LIN {X 0,Y 573.279,Z 329.697,A -85,B 0,C 180,E1 -2325.807,E2 -2325.807} C_VEL
LIN {X 0,Y 573.268,Z 329.699,A -85,B 0,C 180,E1 -2328.745,E2 -2328.745} C_VEL
LIN {X 0,Y 573.26,Z 329.706,A -85,B 0,C 180,E1 -2331.54,E2 -2331.54} C_VEL
LIN {X 0,Y 573.246,Z 329.702,A -85,B 0,C 180,E1 -2333.665,E2 -2333.665} C_VEL
LIN {X 0,Y 573.226,Z 329.704,A -85,B 0,C 180,E1 -2335.781,E2 -2335.781} C_VEL
LIN {X 0,Y 573.314,Z 329.695,A -85,B 0,C 180,E1 -2337.893,E2 -2337.893} C_VEL
LIN {X 0,Y 573.335,Z 329.689,A -85,B 0,C 180,E1 -2340.702,E2 -2340.702} C_VEL
LIN {X 0,Y 573.237,Z 329.705,A -85,B 0,C 180,E1 -2343.515,E2 -2343.515} C_VEL
LIN {X 0,Y 573.295,Z 329.695,A -85,B 0,C 180,E1 -2345.628,E2 -2345.628} C_VEL
LIN {X 0,Y 573.277,Z 329.698,A -85,B 0,C 180,E1 -2347.75,E2 -2347.75} C_VEL
LIN {X 0,Y 573.271,Z 329.698,A -85,B 0,C 180,E1 -2350.597,E2 -2350.597} C_VEL
LIN {X 0,Y 573.269,Z 329.699,A -85,B 0,C 180,E1 -2352.749,E2 -2352.749} C_VEL
LIN {X 0,Y 573.241,Z 329.707,A -85,B 0,C 180,E1 -2354.92,E2 -2354.92} C_VEL
LIN {X 0,Y 573.249,Z 329.701,A -85,B 0,C 180,E1 -2357.848,E2 -2357.848} C_VEL
LIN {X 0,Y 573.246,Z 329.708,A -85,B 0,C 180,E1 -2360.077,E2 -2360.077} C_VEL
LIN {X 0,Y 573.24,Z 329.703,A -85,B 0,C 180,E1 -2362.338,E2 -2362.338} C_VEL
LIN {X 0,Y 573.255,Z 329.699,A -85,B 0,C 180,E1 -2364.389,E2 -2364.389} C_VEL
LIN {X 0,Y 572.629,Z 329.784,A -85,B 0,C 180,E1 -2364.976,E2 -2364.976} C_VEL
LIN {X 0,Y 569.786,Z 330.135,A -85,B 0,C 180,E1 -2365.927,E2 -2365.927} C_VEL
LIN {X 0,Y 567.354,Z 330.441,A -85,B 0,C 180,E1 -2366.693,E2 -2366.693} C_VEL
LIN {X 0,Y 566.298,Z 330.568,A -85,B 0,C 180,E1 -2367.284,E2 -2367.284} C_VEL
LIN {X 0,Y 566.208,Z 330.578,A -85,B 0,C 180,E1 -2367.484,E2 -2367.484} C_VEL
LIN {X 0,Y 566.206,Z 330.58,A -85,B 0,C 180,E1 -2369.769,E2 -2369.769} C_VEL
LIN {X 0,Y 566.207,Z 330.579,A -85,B 0,C 180,E1 -2372.43,E2 -2372.43} C_VEL
LIN {X 0,Y 566.186,Z 330.585,A -85,B 0,C 180,E1 -2374.99,E2 -2374.99} C_VEL
LIN {X 0,Y 566.2,Z 330.58,A -85,B 0,C 180,E1 -2377.461,E2 -2377.461} C_VEL
LIN {X 0,Y 566.211,Z 330.584,A -85,B 0,C 180,E1 -2380.199,E2 -2380.199} C_VEL
LIN {X 0,Y 566.205,Z 330.579,A -85,B 0,C 180,E1 -2383.054,E2 -2383.054} C_VEL
LIN {X 0,Y 566.203,Z 330.58,A -85,B 0,C 180,E1 -2386.049,E2 -2386.049} C_VEL
LIN {X 0,Y 566.186,Z 330.586,A -85,B 0,C 180,E1 -2388.861,E2 -2388.861} C_VEL
LIN {X 0,Y 566.274,Z 330.749,A -85,B 0,C 180,E1 -2391.305,E2 -2391.305} C_VEL
LIN {X 0,Y 566.32,Z 335.336,A -85,B 0,C 180,E1 -2393.77,E2 -2393.77} C_VEL
LIN {X 0,Y 566.259,Z 339.965,A -85,B 0,C 180,E1 -2396.259,E2 -2396.259} C_VEL
LIN {X 0,Y 566.185,Z 344.997,A -85,B 0,C 180,E1 -2398.925,E2 -2398.925} C_VEL
LIN {X 0,Y 566.125,Z 350.67,A -85,B 0,C 180,E1 -2401.852,E2 -2401.852} C_VEL
LIN {X 0,Y 566.061,Z 355.376,A -85,B 0,C 180,E1 -2404.243,E2 -2404.243} C_VEL
LIN {X 0,Y 566.048,Z 360.406,A -85,B 0,C 180,E1 -2406.748,E2 -2406.748} C_VEL
LIN {X 0,Y 566.016,Z 364.889,A -85,B 0,C 180,E1 -2408.895,E2 -2408.895} C_VEL
LIN {X 0,Y 565.984,Z 371.303,A -85,B 0,C 180,E1 -2411.915,E2 -2411.915} C_VEL
LIN {X 0,Y 565.961,Z 377.468,A -85,B 0,C 180,E1 -2414.769,E2 -2414.769} C_VEL
LIN {X 0,Y 567.384,Z 385.385,A -85,B 0,C 180,E1 -2414.949,E2 -2414.949} C_VEL
LIN {X 0,Y 567.258,Z 399.805,A -85,B 0,C 180,E1 -2415.313,E2 -2415.313} C_VEL
LIN {X 0,Y 567.093,Z 414.1,A -85,B 0,C 180,E1 -2415.832,E2 -2415.832} C_VEL
LIN {X 0,Y 566.914,Z 427.265,A -85,B 0,C 180,E1 -2416.468,E2 -2416.468} C_VEL
LIN {X 0,Y 566.715,Z 439.211,A -85,B 0,C 180,E1 -2417.193,E2 -2417.193} C_VEL
LIN {X 0,Y 566.536,Z 451.291,A -85,B 0,C 180,E1 -2418.098,E2 -2418.098} C_VEL
LIN {X 0,Y 566.399,Z 462.502,A -85,B 0,C 180,E1 -2419.126,E2 -2419.126} C_VEL
LIN {X 0,Y 566.202,Z 471.968,A -85,B 0,C 180,E1 -2420.173,E2 -2420.173} C_VEL
LIN {X 0,Y 566.123,Z 480.099,A -85,B 0,C 180,E1 -2421.253,E2 -2421.253} C_VEL
LIN {X 0,Y 566.016,Z 487.881,A -85,B 0,C 180,E1 -2422.509,E2 -2422.509} C_VEL
LIN {X 0,Y 565.945,Z 493.323,A -85,B 0,C 180,E1 -2423.583,E2 -2423.583} C_VEL
LIN {X 0,Y 565.928,Z 497.801,A -85,B 0,C 180,E1 -2424.656,E2 -2424.656} C_VEL
LIN {X 0,Y 565.957,Z 501.311,A -85,B 0,C 180,E1 -2425.727,E2 -2425.727} C_VEL
LIN {X 0,Y 565.875,Z 504.742,A -85,B 0,C 180,E1 -2427.152,E2 -2427.152} C_VEL
LIN {X 0,Y 565.844,Z 506.784,A -85,B 0,C 180,E1 -2428.577,E2 -2428.577} C_VEL
LIN {X 0,Y 565.838,Z 507.496,A -85,B 0,C 180,E1 -2430,E2 -2430} C_VEL
LIN {X 0,Y 565.841,Z 506.881,A -85,B 0,C 180,E1 -2431.424,E2 -2431.424} C_VEL
LIN {X 0,Y 565.873,Z 504.925,A -85,B 0,C 180,E1 -2432.848,E2 -2432.848} C_VEL
LIN {X 0,Y 565.958,Z 501.577,A -85,B 0,C 180,E1 -2434.273,E2 -2434.273} C_VEL
LIN {X 0,Y 565.983,Z 496.745,A -85,B 0,C 180,E1 -2435.701,E2 -2435.701} C_VEL
LIN {X 0,Y 565.981,Z 490.281,A -85,B 0,C 180,E1 -2437.133,E2 -2437.133} C_VEL
LIN {X 0,Y 566.093,Z 483.08,A -85,B 0,C 180,E1 -2438.388,E2 -2438.388} C_VEL
LIN {X 0,Y 566.172,Z 475.539,A -85,B 0,C 180,E1 -2439.467,E2 -2439.467} C_VEL
LIN {X 0,Y 566.29,Z 466.484,A -85,B 0,C 180,E1 -2440.548,E2 -2440.548} C_VEL
LIN {X 0,Y 566.487,Z 457.47,A -85,B 0,C 180,E1 -2441.449,E2 -2441.449} C_VEL
LIN {X 0,Y 566.626,Z 446.716,A -85,B 0,C 180,E1 -2442.354,E2 -2442.354} C_VEL
LIN {X 0,Y 566.767,Z 434.955,A -85,B 0,C 180,E1 -2443.171,E2 -2443.171} C_VEL
LIN {X 0,Y 567.011,Z 421.978,A -85,B 0,C 180,E1 -2443.896,E2 -2443.896} C_VEL
LIN {X 0,Y 567.185,Z 409.289,A -85,B 0,C 180,E1 -2444.451,E2 -2444.451} C_VEL
LIN {X 0,Y 567.306,Z 395.024,A -85,B 0,C 180,E1 -2444.918,E2 -2444.918} C_VEL
LIN {X 0,Y 567.183,Z 383.552,A -85,B 0,C 180,E1 -2445.183,E2 -2445.183} C_VEL
LIN {X 0,Y 565.932,Z 377.463,A -85,B 0,C 180,E1 -2445.324,E2 -2445.324} C_VEL
LIN {X 0,Y 565.976,Z 371.496,A -85,B 0,C 180,E1 -2448.086,E2 -2448.086} C_VEL
LIN {X 0,Y 566.018,Z 365.078,A -85,B 0,C 180,E1 -2451.105,E2 -2451.105} C_VEL
LIN {X 0,Y 566.039,Z 358.692,A -85,B 0,C 180,E1 -2454.188,E2 -2454.188} C_VEL
LIN {X 0,Y 566.084,Z 353.819,A -85,B 0,C 180,E1 -2456.634,E2 -2456.634} C_VEL
LIN {X 0,Y 566.132,Z 349.269,A -85,B 0,C 180,E1 -2458.957,E2 -2458.957} C_VEL
LIN {X 0,Y 566.192,Z 344.506,A -85,B 0,C 180,E1 -2461.422,E2 -2461.422} C_VEL
LIN {X 0,Y 566.258,Z 339.744,A -85,B 0,C 180,E1 -2463.953,E2 -2463.953} C_VEL
LIN {X 0,Y 566.314,Z 334.886,A -85,B 0,C 180,E1 -2466.562,E2 -2466.562} C_VEL
LIN {X 0,Y 566.225,Z 330.582,A -85,B 0,C 180,E1 -2468.893,E2 -2468.893} C_VEL
LIN {X 0,Y 566.193,Z 330.583,A -85,B 0,C 180,E1 -2471.861,E2 -2471.861} C_VEL
LIN {X 0,Y 566.203,Z 330.579,A -85,B 0,C 180,E1 -2474.036,E2 -2474.036} C_VEL
LIN {X 0,Y 566.206,Z 330.578,A -85,B 0,C 180,E1 -2477.083,E2 -2477.083} C_VEL
LIN {X 0,Y 566.221,Z 330.577,A -85,B 0,C 180,E1 -2480.314,E2 -2480.314} C_VEL
LIN {X 0,Y 566.205,Z 330.582,A -85,B 0,C 180,E1 -2483.43,E2 -2483.43} C_VEL
LIN {X 0,Y 566.218,Z 330.58,A -85,B 0,C 180,E1 -2486.266,E2 -2486.266} C_VEL
LIN {X 0,Y 566.196,Z 330.58,A -85,B 0,C 180,E1 -2488.924,E2 -2488.924} C_VEL
LIN {X 0,Y 566.218,Z 330.58,A -85,B 0,C 180,E1 -2491.858,E2 -2491.858} C_VEL
LIN {X 0,Y 566.215,Z 330.577,A -85,B 0,C 180,E1 -2494.251,E2 -2494.251} C_VEL
LIN {X 0,Y 566.179,Z 330.588,A -85,B 0,C 180,E1 -2496.718,E2 -2496.718} C_VEL
LIN {X 0,Y 566.213,Z 330.579,A -85,B 0,C 180,E1 -2499.663,E2 -2499.663} C_VEL
LIN {X 0,Y 566.206,Z 330.578,A -85,B 0,C 180,E1 -2502.668,E2 -2502.668} C_VEL
LIN {X 0,Y 566.236,Z 330.575,A -85,B 0,C 180,E1 -2505.627,E2 -2505.627} C_VEL
LIN {X 0,Y 566.242,Z 330.577,A -85,B 0,C 180,E1 -2508.675,E2 -2508.675} C_VEL
LIN {X 0,Y 566.212,Z 330.58,A -85,B 0,C 180,E1 -2511.434,E2 -2511.434} C_VEL
LIN {X 0,Y 566.263,Z 330.571,A -85,B 0,C 180,E1 -2514.302,E2 -2514.302} C_VEL
LIN {X 0,Y 566.28,Z 330.569,A -85,B 0,C 180,E1 -2517.866,E2 -2517.866} C_VEL
LIN {X 0,Y 566.307,Z 330.566,A -85,B 0,C 180,E1 -2520.711,E2 -2520.711} C_VEL
LIN {X 0,Y 566.277,Z 330.57,A -85,B 0,C 180,E1 -2522.845,E2 -2522.845} C_VEL
LIN {X 0,Y 566.263,Z 330.572,A -85,B 0,C 180,E1 -2525.698,E2 -2525.698} C_VEL
LIN {X 0,Y 566.212,Z 330.584,A -85,B 0,C 180,E1 -2528.566,E2 -2528.566} C_VEL
LIN {X 0,Y 566.249,Z 330.574,A -85,B 0,C 180,E1 -2531.454,E2 -2531.454} C_VEL
LIN {X 0,Y 566.241,Z 330.574,A -85,B 0,C 180,E1 -2534.506,E2 -2534.506} C_VEL
LIN {X 0,Y 566.206,Z 330.581,A -85,B 0,C 180,E1 -2537.331,E2 -2537.331} C_VEL
LIN {X 0,Y 566.213,Z 330.585,A -85,B 0,C 180,E1 -2540.337,E2 -2540.337} C_VEL
LIN {X 0,Y 566.195,Z 330.583,A -85,B 0,C 180,E1 -2543.403,E2 -2543.403} C_VEL
LIN {X 0,Y 566.219,Z 330.579,A -85,B 0,C 180,E1 -2545.749,E2 -2545.749} C_VEL
LIN {X 0,Y 566.208,Z 330.579,A -85,B 0,C 180,E1 -2548.202,E2 -2548.202} C_VEL
LIN {X 0,Y 566.195,Z 330.58,A -85,B 0,C 180,E1 -2551.076,E2 -2551.076} C_VEL
LIN {X 0,Y 566.217,Z 330.584,A -85,B 0,C 180,E1 -2553.734,E2 -2553.734} C_VEL
LIN {X 0,Y 566.22,Z 330.578,A -85,B 0,C 180,E1 -2556.568,E2 -2556.568} C_VEL
LIN {X 0,Y 566.22,Z 330.576,A -85,B 0,C 180,E1 -2559.686,E2 -2559.686} C_VEL
LIN {X 0,Y 566.214,Z 330.584,A -85,B 0,C 180,E1 -2562.087,E2 -2562.087} C_VEL
LIN {X 0,Y 566.173,Z 330.584,A -85,B 0,C 180,E1 -2565.036,E2 -2565.036} C_VEL
LIN {X 0,Y 566.218,Z 330.578,A -85,B 0,C 180,E1 -2567.913,E2 -2567.913} C_VEL
LIN {X 0,Y 566.217,Z 330.583,A -85,B 0,C 180,E1 -2570.726,E2 -2570.726} C_VEL
LIN {X 0,Y 566.247,Z 330.784,A -85,B 0,C 180,E1 -2573.534,E2 -2573.534} C_VEL
LIN {X 0,Y 567.061,Z 335.097,A -85,B 0,C 180,E1 -2574.883,E2 -2574.883} C_VEL
LIN {X 0,Y 566.991,Z 342.231,A -85,B 0,C 180,E1 -2576.948,E2 -2576.948} C_VEL
LIN {X 0,Y 566.836,Z 352.746,A -85,B 0,C 180,E1 -2579.858,E2 -2579.858} C_VEL
LIN {X 0,Y 566.665,Z 363.294,A -85,B 0,C 180,E1 -2582.684,E2 -2582.684} C_VEL
LIN {X 0,Y 566.483,Z 373.873,A -85,B 0,C 180,E1 -2585.442,E2 -2585.442} C_VEL
LIN {X 0,Y 566.404,Z 382.902,A -85,B 0,C 180,E1 -2587.762,E2 -2587.762} C_VEL
LIN {X 0,Y 566.295,Z 394.128,A -85,B 0,C 180,E1 -2590.595,E2 -2590.595} C_VEL
LIN {X 0,Y 566.236,Z 400.283,A -85,B 0,C 180,E1 -2592.128,E2 -2592.128} C_VEL
LIN {X 0,Y 567.998,Z 408.781,A -85,B 0,C 180,E1 -2592.315,E2 -2592.315} C_VEL
LIN {X 0,Y 567.88,Z 424.081,A -85,B 0,C 180,E1 -2592.628,E2 -2592.628} C_VEL
LIN {X 0,Y 567.684,Z 439.2,A -85,B 0,C 180,E1 -2593.086,E2 -2593.086} C_VEL
LIN {X 0,Y 567.454,Z 452.815,A -85,B 0,C 180,E1 -2593.634,E2 -2593.634} C_VEL
LIN {X 0,Y 567.232,Z 467.096,A -85,B 0,C 180,E1 -2594.366,E2 -2594.366} C_VEL
LIN {X 0,Y 566.953,Z 480.511,A -85,B 0,C 180,E1 -2595.216,E2 -2595.216} C_VEL
LIN {X 0,Y 566.738,Z 493.158,A -85,B 0,C 180,E1 -2596.189,E2 -2596.189} C_VEL
LIN {X 0,Y 566.546,Z 504.968,A -85,B 0,C 180,E1 -2597.28,E2 -2597.28} C_VEL
LIN {X 0,Y 566.343,Z 514.901,A -85,B 0,C 180,E1 -2598.366,E2 -2598.366} C_VEL
LIN {X 0,Y 566.204,Z 524.619,A -85,B 0,C 180,E1 -2599.631,E2 -2599.631} C_VEL
LIN {X 0,Y 566.079,Z 532.721,A -85,B 0,C 180,E1 -2600.892,E2 -2600.892} C_VEL
LIN {X 0,Y 566.014,Z 539.424,A -85,B 0,C 180,E1 -2602.15,E2 -2602.15} C_VEL
LIN {X 0,Y 565.943,Z 545.606,A -85,B 0,C 180,E1 -2603.583,E2 -2603.583} C_VEL
LIN {X 0,Y 565.867,Z 550.385,A -85,B 0,C 180,E1 -2605.012,E2 -2605.012} C_VEL
LIN {X 0,Y 565.909,Z 553.889,A -85,B 0,C 180,E1 -2606.44,E2 -2606.44} C_VEL
LIN {X 0,Y 565.839,Z 556.192,A -85,B 0,C 180,E1 -2607.864,E2 -2607.864} C_VEL
LIN {X 0,Y 565.839,Z 557.349,A -85,B 0,C 180,E1 -2609.288,E2 -2609.288} C_VEL
LIN {X 0,Y 565.839,Z 557.349,A -85,B 0,C 180,E1 -2610.712,E2 -2610.712} C_VEL
LIN {X 0,Y 565.839,Z 556.191,A -85,B 0,C 180,E1 -2612.135,E2 -2612.135} C_VEL
LIN {X 0,Y 565.909,Z 553.887,A -85,B 0,C 180,E1 -2613.56,E2 -2613.56} C_VEL
LIN {X 0,Y 565.866,Z 550.385,A -85,B 0,C 180,E1 -2614.988,E2 -2614.988} C_VEL
LIN {X 0,Y 565.942,Z 545.609,A -85,B 0,C 180,E1 -2616.417,E2 -2616.417} C_VEL
LIN {X 0,Y 566.014,Z 539.423,A -85,B 0,C 180,E1 -2617.85,E2 -2617.85} C_VEL
LIN {X 0,Y 566.071,Z 531.648,A -85,B 0,C 180,E1 -2619.288,E2 -2619.288} C_VEL
LIN {X 0,Y 566.24,Z 523.369,A -85,B 0,C 180,E1 -2620.549,E2 -2620.549} C_VEL
LIN {X 0,Y 566.367,Z 513.391,A -85,B 0,C 180,E1 -2621.815,E2 -2621.815} C_VEL
LIN {X 0,Y 566.586,Z 503.188,A -85,B 0,C 180,E1 -2622.901,E2 -2622.901} C_VEL
LIN {X 0,Y 566.763,Z 491.018,A -85,B 0,C 180,E1 -2623.993,E2 -2623.993} C_VEL
LIN {X 0,Y 567.041,Z 478.339,A -85,B 0,C 180,E1 -2624.936,E2 -2624.936} C_VEL
LIN {X 0,Y 567.266,Z 465.514,A -85,B 0,C 180,E1 -2625.725,E2 -2625.725} C_VEL
LIN {X 0,Y 567.494,Z 450.83,A -85,B 0,C 180,E1 -2626.457,E2 -2626.457} C_VEL
LIN {X 0,Y 567.721,Z 436.613,A -85,B 0,C 180,E1 -2627.005,E2 -2627.005} C_VEL
LIN {X 0,Y 567.869,Z 422.051,A -85,B 0,C 180,E1 -2627.424,E2 -2627.424} C_VEL
LIN {X 0,Y 567.893,Z 407.611,A -85,B 0,C 180,E1 -2627.706,E2 -2627.706} C_VEL
LIN {X 0,Y 566.243,Z 400.314,A -85,B 0,C 180,E1 -2627.864,E2 -2627.864} C_VEL
LIN {X 0,Y 566.331,Z 388.922,A -85,B 0,C 180,E1 -2630.712,E2 -2630.712} C_VEL
LIN {X 0,Y 566.488,Z 376.883,A -85,B 0,C 180,E1 -2633.779,E2 -2633.779} C_VEL
LIN {X 0,Y 566.614,Z 365.5,A -85,B 0,C 180,E1 -2636.741,E2 -2636.741} C_VEL
LIN {X 0,Y 566.755,Z 355.701,A -85,B 0,C 180,E1 -2639.329,E2 -2639.329} C_VEL
LIN {X 0,Y 566.975,Z 345.213,A -85,B 0,C 180,E1 -2642.209,E2 -2642.209} C_VEL
LIN {X 0,Y 567.084,Z 336.315,A -85,B 0,C 180,E1 -2644.757,E2 -2644.757} C_VEL
LIN {X 0,Y 566.225,Z 330.582,A -85,B 0,C 180,E1 -2646.568,E2 -2646.568} C_VEL
LIN {X 0,Y 566.217,Z 330.583,A -85,B 0,C 180,E1 -2649.686,E2 -2649.686} C_VEL
LIN {X 0,Y 566.217,Z 330.578,A -85,B 0,C 180,E1 -2652.087,E2 -2652.087} C_VEL
LIN {X 0,Y 566.171,Z 330.585,A -85,B 0,C 180,E1 -2655.037,E2 -2655.037} C_VEL
LIN {X 0,Y 566.215,Z 330.579,A -85,B 0,C 180,E1 -2658.137,E2 -2658.137} C_VEL
LIN {X 0,Y 566.225,Z 330.578,A -85,B 0,C 180,E1 -2660.727,E2 -2660.727} C_VEL
LIN {X 0,Y 566.222,Z 330.577,A -85,B 0,C 180,E1 -2663.784,E2 -2663.784} C_VEL
LIN {X 0,Y 566.216,Z 330.584,A -85,B 0,C 180,E1 -2666.266,E2 -2666.266} C_VEL
LIN {X 0,Y 566.194,Z 330.581,A -85,B 0,C 180,E1 -2668.924,E2 -2668.924} C_VEL
LIN {X 0,Y 566.215,Z 330.578,A -85,B 0,C 180,E1 -2671.858,E2 -2671.858} C_VEL
LIN {X 0,Y 566.218,Z 330.579,A -85,B 0,C 180,E1 -2674.251,E2 -2674.251} C_VEL
LIN {X 0,Y 566.196,Z 330.582,A -85,B 0,C 180,E1 -2676.714,E2 -2676.714} C_VEL
LIN {X 0,Y 566.212,Z 330.583,A -85,B 0,C 180,E1 -2679.663,E2 -2679.663} C_VEL
LIN {X 0,Y 566.205,Z 330.58,A -85,B 0,C 180,E1 -2682.669,E2 -2682.669} C_VEL
LIN {X 0,Y 566.24,Z 330.574,A -85,B 0,C 180,E1 -2685.627,E2 -2685.627} C_VEL
LIN {X 0,Y 566.24,Z 330.575,A -85,B 0,C 180,E1 -2688.676,E2 -2688.676} C_VEL
LIN {X 0,Y 566.211,Z 330.584,A -85,B 0,C 180,E1 -2691.434,E2 -2691.434} C_VEL
LIN {X 0,Y 566.263,Z 330.571,A -85,B 0,C 180,E1 -2694.302,E2 -2694.302} C_VEL
LIN {X 0,Y 566.285,Z 330.57,A -85,B 0,C 180,E1 -2697.866,E2 -2697.866} C_VEL
LIN {X 0,Y 566.306,Z 330.565,A -85,B 0,C 180,E1 -2700.711,E2 -2700.711} C_VEL
LIN {X 0,Y 566.277,Z 330.571,A -85,B 0,C 180,E1 -2702.846,E2 -2702.846} C_VEL
LIN {X 0,Y 566.263,Z 330.571,A -85,B 0,C 180,E1 -2705.698,E2 -2705.698} C_VEL
LIN {X 0,Y 566.211,Z 330.581,A -85,B 0,C 180,E1 -2708.566,E2 -2708.566} C_VEL
LIN {X 0,Y 566.248,Z 330.577,A -85,B 0,C 180,E1 -2711.454,E2 -2711.454} C_VEL
LIN {X 0,Y 566.24,Z 330.575,A -85,B 0,C 180,E1 -2714.506,E2 -2714.506} C_VEL
LIN {X 0,Y 566.205,Z 330.578,A -85,B 0,C 180,E1 -2717.332,E2 -2717.332} C_VEL
LIN {X 0,Y 566.212,Z 330.58,A -85,B 0,C 180,E1 -2720.337,E2 -2720.337} C_VEL
LIN {X 0,Y 566.194,Z 330.587,A -85,B 0,C 180,E1 -2723.404,E2 -2723.404} C_VEL
LIN {X 0,Y 566.214,Z 330.578,A -85,B 0,C 180,E1 -2725.749,E2 -2725.749} C_VEL
LIN {X 0,Y 566.208,Z 330.578,A -85,B 0,C 180,E1 -2727.484,E2 -2727.484} C_VEL
LIN {X 0,Y 565.528,Z 330.666,A -85,B 0,C 180,E1 -2728.078,E2 -2728.078} C_VEL
LIN {X 0,Y 562.662,Z 331.023,A -85,B 0,C 180,E1 -2729.041,E2 -2729.041} C_VEL
LIN {X 0,Y 560.252,Z 331.324,A -85,B 0,C 180,E1 -2729.817,E2 -2729.817} C_VEL
LIN {X 0,Y 559.225,Z 331.452,A -85,B 0,C 180,E1 -2730.416,E2 -2730.416} C_VEL
LIN {X 0,Y 559.144,Z 331.459,A -85,B 0,C 180,E1 -2730.618,E2 -2730.618} C_VEL
LIN {X 0,Y 559.17,Z 331.461,A -85,B 0,C 180,E1 -2733.575,E2 -2733.575} C_VEL
LIN {X 0,Y 559.151,Z 331.459,A -85,B 0,C 180,E1 -2736.445,E2 -2736.445} C_VEL
LIN {X 0,Y 559.179,Z 331.456,A -85,B 0,C 180,E1 -2738.934,E2 -2738.934} C_VEL
LIN {X 0,Y 559.167,Z 331.461,A -85,B 0,C 180,E1 -2741.77,E2 -2741.77} C_VEL
LIN {X 0,Y 559.144,Z 331.46,A -85,B 0,C 180,E1 -2744.739,E2 -2744.739} C_VEL
LIN {X 0,Y 559.181,Z 331.455,A -85,B 0,C 180,E1 -2747.863,E2 -2747.863} C_VEL
LIN {X 0,Y 559.222,Z 331.589,A -85,B 0,C 180,E1 -2751.186,E2 -2751.186} C_VEL
LIN {X 0,Y 559.287,Z 336.402,A -85,B 0,C 180,E1 -2753.8,E2 -2753.8} C_VEL
LIN {X 0,Y 559.207,Z 341.235,A -85,B 0,C 180,E1 -2756.428,E2 -2756.428} C_VEL
LIN {X 0,Y 559.149,Z 346.007,A -85,B 0,C 180,E1 -2758.98,E2 -2758.98} C_VEL
LIN {X 0,Y 559.073,Z 352.333,A -85,B 0,C 180,E1 -2762.282,E2 -2762.282} C_VEL
LIN {X 0,Y 559.019,Z 357.368,A -85,B 0,C 180,E1 -2764.849,E2 -2764.849} C_VEL
LIN {X 0,Y 558.948,Z 363.315,A -85,B 0,C 180,E1 -2767.839,E2 -2767.839} C_VEL
LIN {X 0,Y 558.908,Z 369.701,A -85,B 0,C 180,E1 -2770.917,E2 -2770.917} C_VEL
LIN {X 0,Y 558.884,Z 374.512,A -85,B 0,C 180,E1 -2773.188,E2 -2773.188} C_VEL
LIN {X 0,Y 558.882,Z 377.469,A -85,B 0,C 180,E1 -2774.571,E2 -2774.571} C_VEL
LIN {X 0,Y 560.522,Z 386.231,A -85,B 0,C 180,E1 -2774.777,E2 -2774.777} C_VEL
LIN {X 0,Y 560.388,Z 400.196,A -85,B 0,C 180,E1 -2775.14,E2 -2775.14} C_VEL
LIN {X 0,Y 560.21,Z 414.115,A -85,B 0,C 180,E1 -2775.654,E2 -2775.654} C_VEL
LIN {X 0,Y 560,Z 427.276,A -85,B 0,C 180,E1 -2776.297,E2 -2776.297} C_VEL
LIN {X 0,Y 559.76,Z 439.219,A -85,B 0,C 180,E1 -2777.031,E2 -2777.031} C_VEL
LIN {X 0,Y 559.558,Z 451.296,A -85,B 0,C 180,E1 -2777.947,E2 -2777.947} C_VEL
LIN {X 0,Y 559.417,Z 461.299,A -85,B 0,C 180,E1 -2778.864,E2 -2778.864} C_VEL
LIN {X 0,Y 559.201,Z 470.486,A -85,B 0,C 180,E1 -2779.866,E2 -2779.866} C_VEL
LIN {X 0,Y 559.071,Z 478.867,A -85,B 0,C 180,E1 -2780.959,E2 -2780.959} C_VEL
LIN {X 0,Y 558.973,Z 486.875,A -85,B 0,C 180,E1 -2782.232,E2 -2782.232} C_VEL
LIN {X 0,Y 558.873,Z 493.326,A -85,B 0,C 180,E1 -2783.501,E2 -2783.501} C_VEL
LIN {X 0,Y 558.859,Z 497.803,A -85,B 0,C 180,E1 -2784.588,E2 -2784.588} C_VEL
LIN {X 0,Y 558.866,Z 501.313,A -85,B 0,C 180,E1 -2785.673,E2 -2785.673} C_VEL
LIN {X 0,Y 558.796,Z 504.744,A -85,B 0,C 180,E1 -2787.116,E2 -2787.116} C_VEL
LIN {X 0,Y 558.744,Z 506.785,A -85,B 0,C 180,E1 -2788.559,E2 -2788.559} C_VEL
LIN {X 0,Y 558.739,Z 507.496,A -85,B 0,C 180,E1 -2790,E2 -2790} C_VEL
LIN {X 0,Y 558.741,Z 506.881,A -85,B 0,C 180,E1 -2791.442,E2 -2791.442} C_VEL
LIN {X 0,Y 558.794,Z 504.925,A -85,B 0,C 180,E1 -2792.884,E2 -2792.884} C_VEL
LIN {X 0,Y 558.867,Z 501.576,A -85,B 0,C 180,E1 -2794.327,E2 -2794.327} C_VEL
LIN {X 0,Y 558.912,Z 496.743,A -85,B 0,C 180,E1 -2795.774,E2 -2795.774} C_VEL
LIN {X 0,Y 558.908,Z 490.279,A -85,B 0,C 180,E1 -2797.224,E2 -2797.224} C_VEL
LIN {X 0,Y 559.029,Z 483.077,A -85,B 0,C 180,E1 -2798.495,E2 -2798.495} C_VEL
LIN {X 0,Y 559.124,Z 475.535,A -85,B 0,C 180,E1 -2799.587,E2 -2799.587} C_VEL
LIN {X 0,Y 559.288,Z 466.479,A -85,B 0,C 180,E1 -2800.682,E2 -2800.682} C_VEL
LIN {X 0,Y 559.482,Z 455.508,A -85,B 0,C 180,E1 -2801.779,E2 -2801.779} C_VEL
LIN {X 0,Y 559.669,Z 444.331,A -85,B 0,C 180,E1 -2802.695,E2 -2802.695} C_VEL
LIN {X 0,Y 559.91,Z 431.98,A -85,B 0,C 180,E1 -2803.52,E2 -2803.52} C_VEL
LIN {X 0,Y 560.119,Z 420.092,A -85,B 0,C 180,E1 -2804.163,E2 -2804.163} C_VEL
LIN {X 0,Y 560.359,Z 407.004,A -85,B 0,C 180,E1 -2804.717,E2 -2804.717} C_VEL
LIN {X 0,Y 560.454,Z 393.374,A -85,B 0,C 180,E1 -2805.146,E2 -2805.146} C_VEL
LIN {X 0,Y 560.41,Z 384.975,A -85,B 0,C 180,E1 -2805.341,E2 -2805.341} C_VEL
LIN {X 0,Y 558.877,Z 377.461,A -85,B 0,C 180,E1 -2805.523,E2 -2805.523} C_VEL
LIN {X 0,Y 558.891,Z 371.495,A -85,B 0,C 180,E1 -2808.323,E2 -2808.323} C_VEL
LIN {X 0,Y 558.964,Z 364.839,A -85,B 0,C 180,E1 -2811.499,E2 -2811.499} C_VEL
LIN {X 0,Y 558.984,Z 358.81,A -85,B 0,C 180,E1 -2814.513,E2 -2814.513} C_VEL
LIN {X 0,Y 559.026,Z 354.104,A -85,B 0,C 180,E1 -2816.91,E2 -2816.91} C_VEL
LIN {X 0,Y 559.078,Z 349.35,A -85,B 0,C 180,E1 -2819.358,E2 -2819.358} C_VEL
LIN {X 0,Y 559.169,Z 344.588,A -85,B 0,C 180,E1 -2821.863,E2 -2821.863} C_VEL
LIN {X 0,Y 559.229,Z 339.81,A -85,B 0,C 180,E1 -2824.439,E2 -2824.439} C_VEL
LIN {X 0,Y 559.309,Z 334.905,A -85,B 0,C 180,E1 -2827.096,E2 -2827.096} C_VEL
LIN {X 0,Y 559.187,Z 331.459,A -85,B 0,C 180,E1 -2829.049,E2 -2829.049} C_VEL
LIN {X 0,Y 559.16,Z 331.458,A -85,B 0,C 180,E1 -2832.135,E2 -2832.135} C_VEL
LIN {X 0,Y 559.144,Z 331.465,A -85,B 0,C 180,E1 -2834.739,E2 -2834.739} C_VEL
LIN {X 0,Y 559.16,Z 331.459,A -85,B 0,C 180,E1 -2837.865,E2 -2837.865} C_VEL
LIN {X 0,Y 559.185,Z 331.455,A -85,B 0,C 180,E1 -2840.135,E2 -2840.135} C_VEL
LIN {X 0,Y 559.146,Z 331.46,A -85,B 0,C 180,E1 -2842.892,E2 -2842.892} C_VEL
LIN {X 0,Y 559.172,Z 331.456,A -85,B 0,C 180,E1 -2846.051,E2 -2846.051} C_VEL
LIN {X 0,Y 559.161,Z 331.456,A -85,B 0,C 180,E1 -2848.981,E2 -2848.981} C_VEL
LIN {X 0,Y 559.175,Z 331.461,A -85,B 0,C 180,E1 -2851.619,E2 -2851.619} C_VEL
LIN {X 0,Y 559.184,Z 331.453,A -85,B 0,C 180,E1 -2853.903,E2 -2853.903} C_VEL
LIN {X 0,Y 559.149,Z 331.463,A -85,B 0,C 180,E1 -2856.571,E2 -2856.571} C_VEL
LIN {X 0,Y 559.182,Z 331.453,A -85,B 0,C 180,E1 -2859.395,E2 -2859.395} C_VEL
LIN {X 0,Y 559.148,Z 331.463,A -85,B 0,C 180,E1 -2861.686,E2 -2861.686} C_VEL
LIN {X 0,Y 559.173,Z 331.455,A -85,B 0,C 180,E1 -2863.948,E2 -2863.948} C_VEL
LIN {X 0,Y 559.174,Z 331.455,A -85,B 0,C 180,E1 -2866.184,E2 -2866.184} C_VEL
LIN {X 0,Y 559.213,Z 331.453,A -85,B 0,C 180,E1 -2868.605,E2 -2868.605} C_VEL
LIN {X 0,Y 559.177,Z 331.455,A -85,B 0,C 180,E1 -2871.325,E2 -2871.325} C_VEL
LIN {X 0,Y 559.232,Z 331.446,A -85,B 0,C 180,E1 -2874.23,E2 -2874.23} C_VEL
LIN {X 0,Y 559.245,Z 331.448,A -85,B 0,C 180,E1 -2877.119,E2 -2877.119} C_VEL
LIN {X 0,Y 559.267,Z 331.448,A -85,B 0,C 180,E1 -2880,E2 -2880} C_VEL
LIN {X 0,Y 559.243,Z 331.446,A -85,B 0,C 180,E1 -2882.881,E2 -2882.881} C_VEL
LIN {X 0,Y 559.233,Z 331.448,A -85,B 0,C 180,E1 -2885.77,E2 -2885.77} C_VEL
LIN {X 0,Y 559.176,Z 331.46,A -85,B 0,C 180,E1 -2888.674,E2 -2888.674} C_VEL
LIN {X 0,Y 559.212,Z 331.452,A -85,B 0,C 180,E1 -2891.6,E2 -2891.6} C_VEL
LIN {X 0,Y 559.207,Z 331.451,A -85,B 0,C 180,E1 -2894.595,E2 -2894.595} C_VEL
LIN {X 0,Y 559.165,Z 331.457,A -85,B 0,C 180,E1 -2897.557,E2 -2897.557} C_VEL
LIN {X 0,Y 559.171,Z 331.456,A -85,B 0,C 180,E1 -2899.837,E2 -2899.837} C_VEL
LIN {X 0,Y 559.146,Z 331.462,A -85,B 0,C 180,E1 -2902.152,E2 -2902.152} C_VEL
LIN {X 0,Y 559.185,Z 331.458,A -85,B 0,C 180,E1 -2905.187,E2 -2905.187} C_VEL
LIN {X 0,Y 559.162,Z 331.456,A -85,B 0,C 180,E1 -2907.713,E2 -2907.713} C_VEL
LIN {X 0,Y 559.158,Z 331.46,A -85,B 0,C 180,E1 -2910.182,E2 -2910.182} C_VEL
LIN {X 0,Y 559.16,Z 331.457,A -85,B 0,C 180,E1 -2912.715,E2 -2912.715} C_VEL
LIN {X 0,Y 559.161,Z 331.462,A -85,B 0,C 180,E1 -2915.322,E2 -2915.322} C_VEL
LIN {X 0,Y 559.137,Z 331.46,A -85,B 0,C 180,E1 -2918.017,E2 -2918.017} C_VEL
LIN {X 0,Y 559.161,Z 331.459,A -85,B 0,C 180,E1 -2920.812,E2 -2920.812} C_VEL
LIN {X 0,Y 559.148,Z 331.46,A -85,B 0,C 180,E1 -2923.196,E2 -2923.196} C_VEL
LIN {X 0,Y 559.166,Z 331.457,A -85,B 0,C 180,E1 -2926.268,E2 -2926.268} C_VEL
LIN {X 0,Y 559.164,Z 331.461,A -85,B 0,C 180,E1 -2929.188,E2 -2929.188} C_VEL
LIN {X 0,Y 559.136,Z 331.466,A -85,B 0,C 180,E1 -2931.982,E2 -2931.982} C_VEL
LIN {X 0,Y 559.201,Z 331.613,A -85,B 0,C 180,E1 -2933.251,E2 -2933.251} C_VEL
LIN {X 0,Y 560.071,Z 336.269,A -85,B 0,C 180,E1 -2934.744,E2 -2934.744} C_VEL
LIN {X 0,Y 560.14,Z 342.182,A -85,B 0,C 180,E1 -2936.491,E2 -2936.491} C_VEL
LIN {X 0,Y 559.902,Z 352.673,A -85,B 0,C 180,E1 -2939.445,E2 -2939.445} C_VEL
LIN {X 0,Y 559.687,Z 363.217,A -85,B 0,C 180,E1 -2942.315,E2 -2942.315} C_VEL
LIN {X 0,Y 559.528,Z 373.89,A -85,B 0,C 180,E1 -2945.122,E2 -2945.122} C_VEL
LIN {X 0,Y 559.394,Z 384.407,A -85,B 0,C 180,E1 -2947.857,E2 -2947.857} C_VEL
LIN {X 0,Y 559.231,Z 396.446,A -85,B 0,C 180,E1 -2950.928,E2 -2950.928} C_VEL
LIN {X 0,Y 559.203,Z 400.283,A -85,B 0,C 180,E1 -2951.896,E2 -2951.896} C_VEL
LIN {X 0,Y 561.251,Z 409.999,A -85,B 0,C 180,E1 -2952.115,E2 -2952.115} C_VEL
LIN {X 0,Y 561.074,Z 425.451,A -85,B 0,C 180,E1 -2952.446,E2 -2952.446} C_VEL
LIN {X 0,Y 560.848,Z 440.74,A -85,B 0,C 180,E1 -2952.929,E2 -2952.929} C_VEL
LIN {X 0,Y 560.604,Z 454.799,A -85,B 0,C 180,E1 -2953.522,E2 -2953.522} C_VEL
LIN {X 0,Y 560.317,Z 468.675,A -85,B 0,C 180,E1 -2954.262,E2 -2954.262} C_VEL
LIN {X 0,Y 560.043,Z 481.173,A -85,B 0,C 180,E1 -2955.077,E2 -2955.077} C_VEL
LIN {X 0,Y 559.77,Z 494.226,A -85,B 0,C 180,E1 -2956.106,E2 -2956.106} C_VEL
LIN {X 0,Y 559.558,Z 504.967,A -85,B 0,C 180,E1 -2957.118,E2 -2957.118} C_VEL
LIN {X 0,Y 559.322,Z 514.901,A -85,B 0,C 180,E1 -2958.218,E2 -2958.218} C_VEL
LIN {X 0,Y 559.173,Z 524.62,A -85,B 0,C 180,E1 -2959.499,E2 -2959.499} C_VEL
LIN {X 0,Y 559.026,Z 532.722,A -85,B 0,C 180,E1 -2960.776,E2 -2960.776} C_VEL
LIN {X 0,Y 558.95,Z 539.424,A -85,B 0,C 180,E1 -2962.05,E2 -2962.05} C_VEL
LIN {X 0,Y 558.871,Z 545.606,A -85,B 0,C 180,E1 -2963.501,E2 -2963.501} C_VEL
LIN {X 0,Y 558.787,Z 550.385,A -85,B 0,C 180,E1 -2964.949,E2 -2964.949} C_VEL
LIN {X 0,Y 558.818,Z 553.889,A -85,B 0,C 180,E1 -2966.395,E2 -2966.395} C_VEL
LIN {X 0,Y 558.745,Z 556.191,A -85,B 0,C 180,E1 -2967.837,E2 -2967.837} C_VEL
LIN {X 0,Y 558.739,Z 557.349,A -85,B 0,C 180,E1 -2969.279,E2 -2969.279} C_VEL
LIN {X 0,Y 558.739,Z 557.348,A -85,B 0,C 180,E1 -2970.721,E2 -2970.721} C_VEL
LIN {X 0,Y 558.745,Z 556.19,A -85,B 0,C 180,E1 -2972.162,E2 -2972.162} C_VEL
LIN {X 0,Y 558.818,Z 553.887,A -85,B 0,C 180,E1 -2973.605,E2 -2973.605} C_VEL
LIN {X 0,Y 558.787,Z 550.386,A -85,B 0,C 180,E1 -2975.051,E2 -2975.051} C_VEL
LIN {X 0,Y 558.871,Z 545.609,A -85,B 0,C 180,E1 -2976.499,E2 -2976.499} C_VEL
LIN {X 0,Y 558.95,Z 539.422,A -85,B 0,C 180,E1 -2977.95,E2 -2977.95} C_VEL
LIN {X 0,Y 559.005,Z 531.647,A -85,B 0,C 180,E1 -2979.407,E2 -2979.407} C_VEL
LIN {X 0,Y 559.218,Z 523.368,A -85,B 0,C 180,E1 -2980.683,E2 -2980.683} C_VEL
LIN {X 0,Y 559.362,Z 513.391,A -85,B 0,C 180,E1 -2981.965,E2 -2981.965} C_VEL
LIN {X 0,Y 559.596,Z 503.187,A -85,B 0,C 180,E1 -2983.065,E2 -2983.065} C_VEL
LIN {X 0,Y 559.825,Z 491.019,A -85,B 0,C 180,E1 -2984.17,E2 -2984.17} C_VEL
LIN {X 0,Y 560.125,Z 478.69,A -85,B 0,C 180,E1 -2985.1,E2 -2985.1} C_VEL
LIN {X 0,Y 560.386,Z 465.512,A -85,B 0,C 180,E1 -2985.923,E2 -2985.923} C_VEL
LIN {X 0,Y 560.67,Z 450.827,A -85,B 0,C 180,E1 -2986.663,E2 -2986.663} C_VEL
LIN {X 0,Y 560.96,Z 435.66,A -85,B 0,C 180,E1 -2987.251,E2 -2987.251} C_VEL
LIN {X 0,Y 561.139,Z 420.146,A -85,B 0,C 180,E1 -2987.689,E2 -2987.689} C_VEL
LIN {X 0,Y 561.077,Z 408.432,A -85,B 0,C 180,E1 -2987.916,E2 -2987.916} C_VEL
LIN {X 0,Y 559.186,Z 400.27,A -85,B 0,C 180,E1 -2988.108,E2 -2988.108} C_VEL
LIN {X 0,Y 559.335,Z 388.922,A -85,B 0,C 180,E1 -2990.984,E2 -2990.984} C_VEL
LIN {X 0,Y 559.516,Z 376.883,A -85,B 0,C 180,E1 -2994.094,E2 -2994.094} C_VEL
LIN {X 0,Y 559.696,Z 364.759,A -85,B 0,C 180,E1 -2997.279,E2 -2997.279} C_VEL
LIN {X 0,Y 559.859,Z 354.172,A -85,B 0,C 180,E1 -3000.141,E2 -3000.141} C_VEL
LIN {X 0,Y 560.049,Z 344.739,A -85,B 0,C 180,E1 -3002.778,E2 -3002.778} C_VEL
LIN {X 0,Y 560.149,Z 337.744,A -85,B 0,C 180,E1 -3004.811,E2 -3004.811} C_VEL
LIN {X 0,Y 559.186,Z 331.458,A -85,B 0,C 180,E1 -3006.817,E2 -3006.817} C_VEL
LIN {X 0,Y 559.163,Z 331.459,A -85,B 0,C 180,E1 -3009.942,E2 -3009.942} C_VEL
LIN {X 0,Y 559.167,Z 331.462,A -85,B 0,C 180,E1 -3012.743,E2 -3012.743} C_VEL
LIN {X 0,Y 559.151,Z 331.46,A -85,B 0,C 180,E1 -3015.761,E2 -3015.761} C_VEL
LIN {X 0,Y 559.189,Z 331.453,A -85,B 0,C 180,E1 -3018.232,E2 -3018.232} C_VEL
LIN {X 0,Y 559.181,Z 331.46,A -85,B 0,C 180,E1 -3021.191,E2 -3021.191} C_VEL
LIN {X 0,Y 559.177,Z 331.455,A -85,B 0,C 180,E1 -3023.792,E2 -3023.792} C_VEL
LIN {X 0,Y 559.166,Z 331.461,A -85,B 0,C 180,E1 -3026.425,E2 -3026.425} C_VEL
LIN {X 0,Y 559.158,Z 331.458,A -85,B 0,C 180,E1 -3028.981,E2 -3028.981} C_VEL
LIN {X 0,Y 559.172,Z 331.458,A -85,B 0,C 180,E1 -3031.619,E2 -3031.619} C_VEL
LIN {X 0,Y 559.185,Z 331.453,A -85,B 0,C 180,E1 -3033.903,E2 -3033.903} C_VEL
LIN {X 0,Y 559.161,Z 331.46,A -85,B 0,C 180,E1 -3036.568,E2 -3036.568} C_VEL
LIN {X 0,Y 559.18,Z 331.455,A -85,B 0,C 180,E1 -3039.396,E2 -3039.396} C_VEL
LIN {X 0,Y 559.148,Z 331.46,A -85,B 0,C 180,E1 -3041.686,E2 -3041.686} C_VEL
LIN {X 0,Y 559.17,Z 331.454,A -85,B 0,C 180,E1 -3043.948,E2 -3043.948} C_VEL
LIN {X 0,Y 559.178,Z 331.457,A -85,B 0,C 180,E1 -3046.184,E2 -3046.184} C_VEL
LIN {X 0,Y 559.211,Z 331.451,A -85,B 0,C 180,E1 -3048.605,E2 -3048.605} C_VEL
LIN {X 0,Y 559.175,Z 331.458,A -85,B 0,C 180,E1 -3051.326,E2 -3051.326} C_VEL
LIN {X 0,Y 559.232,Z 331.447,A -85,B 0,C 180,E1 -3054.23,E2 -3054.23} C_VEL
LIN {X 0,Y 559.256,Z 331.445,A -85,B 0,C 180,E1 -3057.84,E2 -3057.84} C_VEL
LIN {X 0,Y 559.276,Z 331.44,A -85,B 0,C 180,E1 -3060.72,E2 -3060.72} C_VEL
LIN {X 0,Y 559.244,Z 331.448,A -85,B 0,C 180,E1 -3062.881,E2 -3062.881} C_VEL
LIN {X 0,Y 559.232,Z 331.447,A -85,B 0,C 180,E1 -3065.77,E2 -3065.77} C_VEL
LIN {X 0,Y 559.176,Z 331.456,A -85,B 0,C 180,E1 -3068.675,E2 -3068.675} C_VEL
LIN {X 0,Y 559.211,Z 331.455,A -85,B 0,C 180,E1 -3071.6,E2 -3071.6} C_VEL
LIN {X 0,Y 559.206,Z 331.452,A -85,B 0,C 180,E1 -3074.596,E2 -3074.596} C_VEL
LIN {X 0,Y 559.164,Z 331.455,A -85,B 0,C 180,E1 -3077.557,E2 -3077.557} C_VEL
LIN {X 0,Y 559.171,Z 331.458,A -85,B 0,C 180,E1 -3079.838,E2 -3079.838} C_VEL
LIN {X 0,Y 559.146,Z 331.46,A -85,B 0,C 180,E1 -3082.153,E2 -3082.153} C_VEL
LIN {X 0,Y 559.18,Z 331.458,A -85,B 0,C 180,E1 -3085.298,E2 -3085.298} C_VEL
LIN {X 0,Y 559.162,Z 331.456,A -85,B 0,C 180,E1 -3087.713,E2 -3087.713} C_VEL
LIN {X 0,Y 559.144,Z 331.459,A -85,B 0,C 180,E1 -3090.618,E2 -3090.618} C_VEL
LIN {X 0,Y 558.483,Z 331.542,A -85,B 0,C 180,E1 -3091.22,E2 -3091.22} C_VEL
LIN {X 0,Y 555.621,Z 331.899,A -85,B 0,C 180,E1 -3092.196,E2 -3092.196} C_VEL
LIN {X 0,Y 553.209,Z 332.198,A -85,B 0,C 180,E1 -3092.981,E2 -3092.981} C_VEL
LIN {X 0,Y 552.189,Z 332.331,A -85,B 0,C 180,E1 -3093.588,E2 -3093.588} C_VEL
LIN {X 0,Y 552.115,Z 332.333,A -85,B 0,C 180,E1 -3093.793,E2 -3093.793} C_VEL
LIN {X 0,Y 552.109,Z 332.34,A -85,B 0,C 180,E1 -3096.747,E2 -3096.747} C_VEL
LIN {X 0,Y 552.134,Z 332.332,A -85,B 0,C 180,E1 -3099.527,E2 -3099.527} C_VEL
LIN {X 0,Y 552.133,Z 332.333,A -85,B 0,C 180,E1 -3102.425,E2 -3102.425} C_VEL
LIN {X 0,Y 552.102,Z 332.34,A -85,B 0,C 180,E1 -3105.563,E2 -3105.563} C_VEL
LIN {X 0,Y 552.133,Z 332.338,A -85,B 0,C 180,E1 -3108.677,E2 -3108.677} C_VEL
LIN {X 0,Y 552.177,Z 332.429,A -85,B 0,C 180,E1 -3111.061,E2 -3111.061} C_VEL
LIN {X 0,Y 552.271,Z 336.481,A -85,B 0,C 180,E1 -3113.295,E2 -3113.295} C_VEL
LIN {X 0,Y 552.208,Z 341.296,A -85,B 0,C 180,E1 -3115.945,E2 -3115.945} C_VEL
LIN {X 0,Y 552.123,Z 346.089,A -85,B 0,C 180,E1 -3118.541,E2 -3118.541} C_VEL
LIN {X 0,Y 552.067,Z 351.574,A -85,B 0,C 180,E1 -3121.449,E2 -3121.449} C_VEL
LIN {X 0,Y 551.967,Z 357.16,A -85,B 0,C 180,E1 -3124.348,E2 -3124.348} C_VEL
LIN {X 0,Y 551.933,Z 361.892,A -85,B 0,C 180,E1 -3126.75,E2 -3126.75} C_VEL
LIN {X 0,Y 551.842,Z 366.563,A -85,B 0,C 180,E1 -3129.109,E2 -3129.109} C_VEL
LIN {X 0,Y 551.808,Z 371.306,A -85,B 0,C 180,E1 -3131.433,E2 -3131.433} C_VEL
LIN {X 0,Y 551.786,Z 377.32,A -85,B 0,C 180,E1 -3134.297,E2 -3134.297} C_VEL
LIN {X 0,Y 551.79,Z 377.471,A -85,B 0,C 180,E1 -3134.368,E2 -3134.368} C_VEL
LIN {X 0,Y 553.668,Z 387.149,A -85,B 0,C 180,E1 -3134.602,E2 -3134.602} C_VEL
LIN {X 0,Y 553.503,Z 401.481,A -85,B 0,C 180,E1 -3134.99,E2 -3134.99} C_VEL
LIN {X 0,Y 553.311,Z 415.203,A -85,B 0,C 180,E1 -3135.519,E2 -3135.519} C_VEL
LIN {X 0,Y 553.036,Z 428.876,A -85,B 0,C 180,E1 -3136.215,E2 -3136.215} C_VEL
LIN {X 0,Y 552.783,Z 440.52,A -85,B 0,C 180,E1 -3136.958,E2 -3136.958} C_VEL
LIN {X 0,Y 552.542,Z 452.37,A -85,B 0,C 180,E1 -3137.885,E2 -3137.885} C_VEL
LIN {X 0,Y 552.398,Z 462.768,A -85,B 0,C 180,E1 -3138.874,E2 -3138.874} C_VEL
LIN {X 0,Y 552.132,Z 471.977,A -85,B 0,C 180,E1 -3139.92,E2 -3139.92} C_VEL
LIN {X 0,Y 552.009,Z 480.105,A -85,B 0,C 180,E1 -3141.027,E2 -3141.027} C_VEL
LIN {X 0,Y 551.902,Z 487.886,A -85,B 0,C 180,E1 -3142.316,E2 -3142.316} C_VEL
LIN {X 0,Y 551.786,Z 494.436,A -85,B 0,C 180,E1 -3143.67,E2 -3143.67} C_VEL
LIN {X 0,Y 551.715,Z 499.049,A -85,B 0,C 180,E1 -3144.884,E2 -3144.884} C_VEL
LIN {X 0,Y 551.741,Z 503.208,A -85,B 0,C 180,E1 -3146.348,E2 -3146.348} C_VEL
LIN {X 0,Y 551.656,Z 505.935,A -85,B 0,C 180,E1 -3147.81,E2 -3147.81} C_VEL
LIN {X 0,Y 551.637,Z 507.306,A -85,B 0,C 180,E1 -3149.27,E2 -3149.27} C_VEL
LIN {X 0,Y 551.638,Z 507.355,A -85,B 0,C 180,E1 -3150.73,E2 -3150.73} C_VEL
LIN {X 0,Y 551.655,Z 506.072,A -85,B 0,C 180,E1 -3152.19,E2 -3152.19} C_VEL
LIN {X 0,Y 551.741,Z 503.428,A -85,B 0,C 180,E1 -3153.652,E2 -3153.652} C_VEL
LIN {X 0,Y 551.715,Z 499.351,A -85,B 0,C 180,E1 -3155.116,E2 -3155.116} C_VEL
LIN {X 0,Y 551.785,Z 494.836,A -85,B 0,C 180,E1 -3156.329,E2 -3156.329} C_VEL
LIN {X 0,Y 551.898,Z 488.382,A -85,B 0,C 180,E1 -3157.684,E2 -3157.684} C_VEL
LIN {X 0,Y 552.002,Z 480.705,A -85,B 0,C 180,E1 -3158.973,E2 -3158.973} C_VEL
LIN {X 0,Y 552.175,Z 471.212,A -85,B 0,C 180,E1 -3160.265,E2 -3160.265} C_VEL
LIN {X 0,Y 552.371,Z 460.858,A -85,B 0,C 180,E1 -3161.416,E2 -3161.416} C_VEL
LIN {X 0,Y 552.624,Z 450.185,A -85,B 0,C 180,E1 -3162.393,E2 -3162.393} C_VEL
LIN {X 0,Y 552.855,Z 439.171,A -85,B 0,C 180,E1 -3163.228,E2 -3163.228} C_VEL
LIN {X 0,Y 553.116,Z 427.222,A -85,B 0,C 180,E1 -3163.97,E2 -3163.97} C_VEL
LIN {X 0,Y 553.276,Z 414.031,A -85,B 0,C 180,E1 -3164.623,E2 -3164.623} C_VEL
LIN {X 0,Y 553.502,Z 400.159,A -85,B 0,C 180,E1 -3165.141,E2 -3165.141} C_VEL
LIN {X 0,Y 553.569,Z 386.186,A -85,B 0,C 180,E1 -3165.51,E2 -3165.51} C_VEL
LIN {X 0,Y 551.765,Z 377.46,A -85,B 0,C 180,E1 -3165.728,E2 -3165.728} C_VEL
LIN {X 0,Y 551.802,Z 373.098,A -85,B 0,C 180,E1 -3167.799,E2 -3167.799} C_VEL
LIN {X 0,Y 551.816,Z 368.298,A -85,B 0,C 180,E1 -3170.113,E2 -3170.113} C_VEL
LIN {X 0,Y 551.895,Z 363.642,A -85,B 0,C 180,E1 -3172.46,E2 -3172.46} C_VEL
LIN {X 0,Y 551.974,Z 358.027,A -85,B 0,C 180,E1 -3175.31,E2 -3175.31} C_VEL
LIN {X 0,Y 552.068,Z 351.738,A -85,B 0,C 180,E1 -3178.551,E2 -3178.551} C_VEL
LIN {X 0,Y 552.115,Z 346.223,A -85,B 0,C 180,E1 -3181.476,E2 -3181.476} C_VEL
LIN {X 0,Y 552.194,Z 341.246,A -85,B 0,C 180,E1 -3184.179,E2 -3184.179} C_VEL
LIN {X 0,Y 552.273,Z 336.585,A -85,B 0,C 180,E1 -3186.735,E2 -3186.735} C_VEL
LIN {X 0,Y 552.233,Z 333.239,A -85,B 0,C 180,E1 -3188.58,E2 -3188.58} C_VEL
LIN {X 0,Y 552.17,Z 332.334,A -85,B 0,C 180,E1 -3189.131,E2 -3189.131} C_VEL
LIN {X 0,Y 552.134,Z 332.333,A -85,B 0,C 180,E1 -3192.426,E2 -3192.426} C_VEL
LIN {X 0,Y 552.101,Z 332.335,A -85,B 0,C 180,E1 -3195.563,E2 -3195.563} C_VEL
LIN {X 0,Y 552.125,Z 332.334,A -85,B 0,C 180,E1 -3198.554,E2 -3198.554} C_VEL
LIN {X 0,Y 552.123,Z 332.338,A -85,B 0,C 180,E1 -3201.411,E2 -3201.411} C_VEL
LIN {X 0,Y 552.091,Z 332.337,A -85,B 0,C 180,E1 -3204.157,E2 -3204.157} C_VEL
LIN {X 0,Y 552.121,Z 332.336,A -85,B 0,C 180,E1 -3206.814,E2 -3206.814} C_VEL
LIN {X 0,Y 552.108,Z 332.336,A -85,B 0,C 180,E1 -3209.391,E2 -3209.391} C_VEL
LIN {X 0,Y 552.116,Z 332.337,A -85,B 0,C 180,E1 -3211.902,E2 -3211.902} C_VEL
LIN {X 0,Y 552.161,Z 332.33,A -85,B 0,C 180,E1 -3214.65,E2 -3214.65} C_VEL
LIN {X 0,Y 552.099,Z 332.336,A -85,B 0,C 180,E1 -3217.549,E2 -3217.549} C_VEL
LIN {X 0,Y 552.151,Z 332.331,A -85,B 0,C 180,E1 -3220.375,E2 -3220.375} C_VEL
LIN {X 0,Y 552.163,Z 332.329,A -85,B 0,C 180,E1 -3222.977,E2 -3222.977} C_VEL
LIN {X 0,Y 552.139,Z 332.331,A -85,B 0,C 180,E1 -3226.004,E2 -3226.004} C_VEL
LIN {X 0,Y 552.169,Z 332.327,A -85,B 0,C 180,E1 -3228.993,E2 -3228.993} C_VEL
LIN {X 0,Y 552.156,Z 332.333,A -85,B 0,C 180,E1 -3231.951,E2 -3231.951} C_VEL
LIN {X 0,Y 552.235,Z 332.322,A -85,B 0,C 180,E1 -3234.889,E2 -3234.889} C_VEL
LIN {X 0,Y 552.224,Z 332.32,A -85,B 0,C 180,E1 -3237.812,E2 -3237.812} C_VEL
LIN {X 0,Y 552.248,Z 332.317,A -85,B 0,C 180,E1 -3240.729,E2 -3240.729} C_VEL
LIN {X 0,Y 552.21,Z 332.322,A -85,B 0,C 180,E1 -3242.918,E2 -3242.918} C_VEL
LIN {X 0,Y 552.203,Z 332.323,A -85,B 0,C 180,E1 -3245.844,E2 -3245.844} C_VEL
LIN {X 0,Y 552.148,Z 332.334,A -85,B 0,C 180,E1 -3248.786,E2 -3248.786} C_VEL
LIN {X 0,Y 552.17,Z 332.331,A -85,B 0,C 180,E1 -3251.75,E2 -3251.75} C_VEL
LIN {X 0,Y 552.143,Z 332.331,A -85,B 0,C 180,E1 -3254.748,E2 -3254.748} C_VEL
LIN {X 0,Y 552.115,Z 332.334,A -85,B 0,C 180,E1 -3257.788,E2 -3257.788} C_VEL
LIN {X 0,Y 552.132,Z 332.336,A -85,B 0,C 180,E1 -3260.101,E2 -3260.101} C_VEL
LIN {X 0,Y 552.101,Z 332.337,A -85,B 0,C 180,E1 -3262.45,E2 -3262.45} C_VEL
LIN {X 0,Y 552.161,Z 332.334,A -85,B 0,C 180,E1 -3265.35,E2 -3265.35} C_VEL
LIN {X 0,Y 552.115,Z 332.335,A -85,B 0,C 180,E1 -3268.098,E2 -3268.098} C_VEL
LIN {X 0,Y 552.107,Z 332.339,A -85,B 0,C 180,E1 -3270.609,E2 -3270.609} C_VEL
LIN {X 0,Y 552.12,Z 332.335,A -85,B 0,C 180,E1 -3273.185,E2 -3273.185} C_VEL
LIN {X 0,Y 552.117,Z 332.336,A -85,B 0,C 180,E1 -3275.841,E2 -3275.841} C_VEL
LIN {X 0,Y 552.126,Z 332.336,A -85,B 0,C 180,E1 -3279.061,E2 -3279.061} C_VEL
LIN {X 0,Y 552.134,Z 332.332,A -85,B 0,C 180,E1 -3281.445,E2 -3281.445} C_VEL
LIN {X 0,Y 552.094,Z 332.336,A -85,B 0,C 180,E1 -3284.531,E2 -3284.531} C_VEL
LIN {X 0,Y 552.135,Z 332.335,A -85,B 0,C 180,E1 -3287.584,E2 -3287.584} C_VEL
LIN {X 0,Y 552.132,Z 332.338,A -85,B 0,C 180,E1 -3290.473,E2 -3290.473} C_VEL
LIN {X 0,Y 552.156,Z 332.49,A -85,B 0,C 180,E1 -3292.971,E2 -3292.971} C_VEL
LIN {X 0,Y 553.161,Z 338.062,A -85,B 0,C 180,E1 -3294.785,E2 -3294.785} C_VEL
LIN {X 0,Y 553.194,Z 343.617,A -85,B 0,C 180,E1 -3296.451,E2 -3296.451} C_VEL
LIN {X 0,Y 552.93,Z 354.107,A -85,B 0,C 180,E1 -3299.441,E2 -3299.441} C_VEL
LIN {X 0,Y 552.703,Z 364.664,A -85,B 0,C 180,E1 -3302.346,E2 -3302.346} C_VEL
LIN {X 0,Y 552.498,Z 375.289,A -85,B 0,C 180,E1 -3305.179,E2 -3305.179} C_VEL
LIN {X 0,Y 552.378,Z 385.913,A -85,B 0,C 180,E1 -3307.955,E2 -3307.955} C_VEL
LIN {X 0,Y 552.217,Z 396.446,A -85,B 0,C 180,E1 -3310.676,E2 -3310.676} C_VEL
LIN {X 0,Y 552.138,Z 400.284,A -85,B 0,C 180,E1 -3311.656,E2 -3311.656} C_VEL
LIN {X 0,Y 554.499,Z 410.931,A -85,B 0,C 180,E1 -3311.904,E2 -3311.904} C_VEL
LIN {X 0,Y 554.302,Z 426.595,A -85,B 0,C 180,E1 -3312.254,E2 -3312.254} C_VEL
LIN {X 0,Y 554.06,Z 441.129,A -85,B 0,C 180,E1 -3312.728,E2 -3312.728} C_VEL
LIN {X 0,Y 553.767,Z 454.798,A -85,B 0,C 180,E1 -3313.313,E2 -3313.313} C_VEL
LIN {X 0,Y 553.458,Z 468.674,A -85,B 0,C 180,E1 -3314.062,E2 -3314.062} C_VEL
LIN {X 0,Y 553.127,Z 481.895,A -85,B 0,C 180,E1 -3314.939,E2 -3314.939} C_VEL
LIN {X 0,Y 552.813,Z 494.223,A -85,B 0,C 180,E1 -3315.928,E2 -3315.928} C_VEL
LIN {X 0,Y 552.584,Z 504.966,A -85,B 0,C 180,E1 -3316.953,E2 -3316.953} C_VEL
LIN {X 0,Y 552.32,Z 514.902,A -85,B 0,C 180,E1 -3318.066,E2 -3318.066} C_VEL
LIN {X 0,Y 552.153,Z 524.62,A -85,B 0,C 180,E1 -3319.364,E2 -3319.364} C_VEL
LIN {X 0,Y 551.945,Z 532.722,A -85,B 0,C 180,E1 -3320.657,E2 -3320.657} C_VEL
LIN {X 0,Y 551.876,Z 539.423,A -85,B 0,C 180,E1 -3321.947,E2 -3321.947} C_VEL
LIN {X 0,Y 551.788,Z 545.72,A -85,B 0,C 180,E1 -3323.447,E2 -3323.447} C_VEL
LIN {X 0,Y 551.713,Z 550.386,A -85,B 0,C 180,E1 -3324.884,E2 -3324.884} C_VEL
LIN {X 0,Y 551.73,Z 553.889,A -85,B 0,C 180,E1 -3326.348,E2 -3326.348} C_VEL
LIN {X 0,Y 551.655,Z 556.191,A -85,B 0,C 180,E1 -3327.81,E2 -3327.81} C_VEL
LIN {X 0,Y 551.639,Z 557.349,A -85,B 0,C 180,E1 -3329.27,E2 -3329.27} C_VEL
LIN {X 0,Y 551.639,Z 557.348,A -85,B 0,C 180,E1 -3330.73,E2 -3330.73} C_VEL
LIN {X 0,Y 551.655,Z 556.189,A -85,B 0,C 180,E1 -3332.19,E2 -3332.19} C_VEL
LIN {X 0,Y 551.73,Z 553.886,A -85,B 0,C 180,E1 -3333.652,E2 -3333.652} C_VEL
LIN {X 0,Y 551.713,Z 550.386,A -85,B 0,C 180,E1 -3335.116,E2 -3335.116} C_VEL
LIN {X 0,Y 551.82,Z 545.609,A -85,B 0,C 180,E1 -3336.582,E2 -3336.582} C_VEL
LIN {X 0,Y 551.876,Z 539.422,A -85,B 0,C 180,E1 -3338.053,E2 -3338.053} C_VEL
LIN {X 0,Y 551.95,Z 531.646,A -85,B 0,C 180,E1 -3339.528,E2 -3339.528} C_VEL
LIN {X 0,Y 552.184,Z 523.368,A -85,B 0,C 180,E1 -3340.821,E2 -3340.821} C_VEL
LIN {X 0,Y 552.352,Z 513.391,A -85,B 0,C 180,E1 -3342.119,E2 -3342.119} C_VEL
LIN {X 0,Y 552.609,Z 503.186,A -85,B 0,C 180,E1 -3343.234,E2 -3343.234} C_VEL
LIN {X 0,Y 552.889,Z 491.019,A -85,B 0,C 180,E1 -3344.352,E2 -3344.352} C_VEL
LIN {X 0,Y 553.247,Z 478.444,A -85,B 0,C 180,E1 -3345.31,E2 -3345.31} C_VEL
LIN {X 0,Y 553.527,Z 465.509,A -85,B 0,C 180,E1 -3346.126,E2 -3346.126} C_VEL
LIN {X 0,Y 553.869,Z 450.825,A -85,B 0,C 180,E1 -3346.874,E2 -3346.874} C_VEL
LIN {X 0,Y 554.161,Z 436.318,A -85,B 0,C 180,E1 -3347.445,E2 -3347.445} C_VEL
LIN {X 0,Y 554.338,Z 422.051,A -85,B 0,C 180,E1 -3347.863,E2 -3347.863} C_VEL
LIN {X 0,Y 554.359,Z 409.845,A -85,B 0,C 180,E1 -3348.118,E2 -3348.118} C_VEL
LIN {X 0,Y 552.155,Z 400.292,A -85,B 0,C 180,E1 -3348.341,E2 -3348.341} C_VEL
LIN {X 0,Y 552.319,Z 388.922,A -85,B 0,C 180,E1 -3351.263,E2 -3351.263} C_VEL
LIN {X 0,Y 552.482,Z 378.316,A -85,B 0,C 180,E1 -3354.021,E2 -3354.021} C_VEL
LIN {X 0,Y 552.659,Z 366.721,A -85,B 0,C 180,E1 -3357.106,E2 -3357.106} C_VEL
LIN {X 0,Y 552.902,Z 355.427,A -85,B 0,C 180,E1 -3360.191,E2 -3360.191} C_VEL
LIN {X 0,Y 553.13,Z 345.119,A -85,B 0,C 180,E1 -3363.117,E2 -3363.117} C_VEL
LIN {X 0,Y 553.227,Z 339.177,A -85,B 0,C 180,E1 -3364.867,E2 -3364.867} C_VEL
LIN {X 0,Y 552.156,Z 332.492,A -85,B 0,C 180,E1 -3367.028,E2 -3367.028} C_VEL
LIN {X 0,Y 552.132,Z 332.34,A -85,B 0,C 180,E1 -3369.527,E2 -3369.527} C_VEL
LIN {X 0,Y 552.133,Z 332.334,A -85,B 0,C 180,E1 -3372.426,E2 -3372.426} C_VEL
LIN {X 0,Y 552.096,Z 332.338,A -85,B 0,C 180,E1 -3375.563,E2 -3375.563} C_VEL
LIN {X 0,Y 552.141,Z 332.328,A -85,B 0,C 180,E1 -3378.677,E2 -3378.677} C_VEL
LIN {X 0,Y 552.123,Z 332.338,A -85,B 0,C 180,E1 -3381.412,E2 -3381.412} C_VEL
LIN {X 0,Y 552.117,Z 332.336,A -85,B 0,C 180,E1 -3384.159,E2 -3384.159} C_VEL
LIN {X 0,Y 552.119,Z 332.336,A -85,B 0,C 180,E1 -3386.814,E2 -3386.814} C_VEL
LIN {X 0,Y 552.106,Z 332.34,A -85,B 0,C 180,E1 -3389.391,E2 -3389.391} C_VEL
LIN {X 0,Y 552.113,Z 332.335,A -85,B 0,C 180,E1 -3391.902,E2 -3391.902} C_VEL
LIN {X 0,Y 552.16,Z 332.334,A -85,B 0,C 180,E1 -3394.65,E2 -3394.65} C_VEL
LIN {X 0,Y 552.1,Z 332.337,A -85,B 0,C 180,E1 -3397.549,E2 -3397.549} C_VEL
LIN {X 0,Y 552.156,Z 332.328,A -85,B 0,C 180,E1 -3400.675,E2 -3400.675} C_VEL
LIN {X 0,Y 552.12,Z 332.332,A -85,B 0,C 180,E1 -3403.738,E2 -3403.738} C_VEL
LIN {X 0,Y 552.141,Z 332.332,A -85,B 0,C 180,E1 -3406.005,E2 -3406.005} C_VEL
LIN {X 0,Y 552.166,Z 332.327,A -85,B 0,C 180,E1 -3408.994,E2 -3408.994} C_VEL
LIN {X 0,Y 552.155,Z 332.33,A -85,B 0,C 180,E1 -3411.952,E2 -3411.952} C_VEL
LIN {X 0,Y 552.234,Z 332.326,A -85,B 0,C 180,E1 -3414.889,E2 -3414.889} C_VEL
LIN {X 0,Y 552.228,Z 332.32,A -85,B 0,C 180,E1 -3417.812,E2 -3417.812} C_VEL
LIN {X 0,Y 552.247,Z 332.316,A -85,B 0,C 180,E1 -3420.729,E2 -3420.729} C_VEL
LIN {X 0,Y 552.21,Z 332.324,A -85,B 0,C 180,E1 -3422.918,E2 -3422.918} C_VEL
LIN {X 0,Y 552.202,Z 332.323,A -85,B 0,C 180,E1 -3425.844,E2 -3425.844} C_VEL
LIN {X 0,Y 552.147,Z 332.331,A -85,B 0,C 180,E1 -3428.786,E2 -3428.786} C_VEL
LIN {X 0,Y 552.169,Z 332.333,A -85,B 0,C 180,E1 -3431.751,E2 -3431.751} C_VEL
LIN {X 0,Y 552.143,Z 332.333,A -85,B 0,C 180,E1 -3434.748,E2 -3434.748} C_VEL
LIN {X 0,Y 552.115,Z 332.334,A -85,B 0,C 180,E1 -3437.789,E2 -3437.789} C_VEL
LIN {X 0,Y 552.132,Z 332.338,A -85,B 0,C 180,E1 -3440.101,E2 -3440.101} C_VEL
LIN {X 0,Y 552.098,Z 332.336,A -85,B 0,C 180,E1 -3442.451,E2 -3442.451} C_VEL
LIN {X 0,Y 552.16,Z 332.332,A -85,B 0,C 180,E1 -3445.35,E2 -3445.35} C_VEL
LIN {X 0,Y 552.115,Z 332.336,A -85,B 0,C 180,E1 -3448.098,E2 -3448.098} C_VEL
LIN {X 0,Y 552.107,Z 332.336,A -85,B 0,C 180,E1 -3450.614,E2 -3450.614} C_VEL
LIN {X 0,Y 552.122,Z 332.335,A -85,B 0,C 180,E1 -3453.186,E2 -3453.186} C_VEL
LIN {X 0,Y 552.115,Z 332.333,A -85,B 0,C 180,E1 -3453.793,E2 -3453.793} C_VEL
LIN {X 0,Y 551.48,Z 332.415,A -85,B 0,C 180,E1 -3454.402,E2 -3454.402} C_VEL
LIN {X 0,Y 548.657,Z 332.774,A -85,B 0,C 180,E1 -3455.39,E2 -3455.39} C_VEL
LIN {X 0,Y 546.235,Z 333.078,A -85,B 0,C 180,E1 -3456.185,E2 -3456.185} C_VEL
LIN {X 0,Y 545.167,Z 333.207,A -85,B 0,C 180,E1 -3456.799,E2 -3456.799} C_VEL
LIN {X 0,Y 545.065,Z 333.217,A -85,B 0,C 180,E1 -3457.007,E2 -3457.007} C_VEL
LIN {X 0,Y 545.07,Z 333.217,A -85,B 0,C 180,E1 -3460.142,E2 -3460.142} C_VEL
LIN {X 0,Y 545.083,Z 333.211,A -85,B 0,C 180,E1 -3463.106,E2 -3463.106} C_VEL
LIN {X 0,Y 545.071,Z 333.213,A -85,B 0,C 180,E1 -3466.224,E2 -3466.224} C_VEL
LIN {X 0,Y 545.091,Z 333.214,A -85,B 0,C 180,E1 -3468.886,E2 -3468.886} C_VEL
LIN {X 0,Y 545.115,Z 333.285,A -85,B 0,C 180,E1 -3470.94,E2 -3470.94} C_VEL
LIN {X 0,Y 545.239,Z 338.094,A -85,B 0,C 180,E1 -3473.635,E2 -3473.635} C_VEL
LIN {X 0,Y 545.142,Z 342.962,A -85,B 0,C 180,E1 -3476.333,E2 -3476.333} C_VEL
LIN {X 0,Y 545.056,Z 347.759,A -85,B 0,C 180,E1 -3478.951,E2 -3478.951} C_VEL
LIN {X 0,Y 545.011,Z 352.526,A -85,B 0,C 180,E1 -3481.502,E2 -3481.502} C_VEL
LIN {X 0,Y 544.911,Z 358.305,A -85,B 0,C 180,E1 -3484.532,E2 -3484.532} C_VEL
LIN {X 0,Y 544.843,Z 363.583,A -85,B 0,C 180,E1 -3487.234,E2 -3487.234} C_VEL
LIN {X 0,Y 544.763,Z 368.265,A -85,B 0,C 180,E1 -3489.615,E2 -3489.615} C_VEL
LIN {X 0,Y 544.738,Z 374.515,A -85,B 0,C 180,E1 -3492.738,E2 -3492.738} C_VEL
LIN {X 0,Y 544.706,Z 377.677,A -85,B 0,C 180,E1 -3494.165,E2 -3494.165} C_VEL
LIN {X 0,Y 546.827,Z 388.52,A -85,B 0,C 180,E1 -3494.433,E2 -3494.433} C_VEL
LIN {X 0,Y 546.636,Z 402.788,A -85,B 0,C 180,E1 -3494.842,E2 -3494.842} C_VEL
LIN {X 0,Y 546.415,Z 416.207,A -85,B 0,C 180,E1 -3495.379,E2 -3495.379} C_VEL
LIN {X 0,Y 546.127,Z 428.884,A -85,B 0,C 180,E1 -3496.037,E2 -3496.037} C_VEL
LIN {X 0,Y 545.82,Z 441.817,A -85,B 0,C 180,E1 -3496.883,E2 -3496.883} C_VEL
LIN {X 0,Y 545.552,Z 453.444,A -85,B 0,C 180,E1 -3497.822,E2 -3497.822} C_VEL
LIN {X 0,Y 545.339,Z 463.967,A -85,B 0,C 180,E1 -3498.854,E2 -3498.854} C_VEL
LIN {X 0,Y 545.091,Z 473.466,A -85,B 0,C 180,E1 -3499.976,E2 -3499.976} C_VEL
LIN {X 0,Y 544.911,Z 482.53,A -85,B 0,C 180,E1 -3501.283,E2 -3501.283} C_VEL
LIN {X 0,Y 544.785,Z 489.833,A -85,B 0,C 180,E1 -3502.588,E2 -3502.588} C_VEL
LIN {X 0,Y 544.732,Z 496.396,A -85,B 0,C 180,E1 -3504.076,E2 -3504.076} C_VEL
LIN {X 0,Y 544.654,Z 501.316,A -85,B 0,C 180,E1 -3505.56,E2 -3505.56} C_VEL
LIN {X 0,Y 544.647,Z 504.746,A -85,B 0,C 180,E1 -3507.041,E2 -3507.041} C_VEL
LIN {X 0,Y 544.544,Z 506.787,A -85,B 0,C 180,E1 -3508.521,E2 -3508.521} C_VEL
LIN {X 0,Y 544.54,Z 507.496,A -85,B 0,C 180,E1 -3510,E2 -3510} C_VEL
LIN {X 0,Y 544.542,Z 506.88,A -85,B 0,C 180,E1 -3511.479,E2 -3511.479} C_VEL
LIN {X 0,Y 544.646,Z 504.924,A -85,B 0,C 180,E1 -3512.959,E2 -3512.959} C_VEL
LIN {X 0,Y 544.655,Z 501.573,A -85,B 0,C 180,E1 -3514.44,E2 -3514.44} C_VEL
LIN {X 0,Y 544.73,Z 496.738,A -85,B 0,C 180,E1 -3515.924,E2 -3515.924} C_VEL
LIN {X 0,Y 544.784,Z 490.274,A -85,B 0,C 180,E1 -3517.412,E2 -3517.412} C_VEL
LIN {X 0,Y 544.906,Z 483.071,A -85,B 0,C 180,E1 -3518.717,E2 -3518.717} C_VEL
LIN {X 0,Y 545.04,Z 475.526,A -85,B 0,C 180,E1 -3519.837,E2 -3519.837} C_VEL
LIN {X 0,Y 545.277,Z 466.468,A -85,B 0,C 180,E1 -3520.959,E2 -3520.959} C_VEL
LIN {X 0,Y 545.506,Z 455.494,A -85,B 0,C 180,E1 -3522.085,E2 -3522.085} C_VEL
LIN {X 0,Y 545.777,Z 444.316,A -85,B 0,C 180,E1 -3523.024,E2 -3523.024} C_VEL
LIN {X 0,Y 546.064,Z 431.965,A -85,B 0,C 180,E1 -3523.87,E2 -3523.87} C_VEL
LIN {X 0,Y 546.315,Z 420.071,A -85,B 0,C 180,E1 -3524.528,E2 -3524.528} C_VEL
LIN {X 0,Y 546.632,Z 407.871,A -85,B 0,C 180,E1 -3525.062,E2 -3525.062} C_VEL
LIN {X 0,Y 546.773,Z 394.226,A -85,B 0,C 180,E1 -3525.511,E2 -3525.511} C_VEL
LIN {X 0,Y 546.712,Z 387.099,A -85,B 0,C 180,E1 -3525.69,E2 -3525.69} C_VEL
LIN {X 0,Y 544.699,Z 377.459,A -85,B 0,C 180,E1 -3525.937,E2 -3525.937} C_VEL
LIN {X 0,Y 544.715,Z 373.122,A -85,B 0,C 180,E1 -3528.038,E2 -3528.038} C_VEL
LIN {X 0,Y 544.764,Z 368.443,A -85,B 0,C 180,E1 -3530.385,E2 -3530.385} C_VEL
LIN {X 0,Y 544.843,Z 363.762,A -85,B 0,C 180,E1 -3532.767,E2 -3532.767} C_VEL
LIN {X 0,Y 544.912,Z 358.507,A -85,B 0,C 180,E1 -3535.468,E2 -3535.468} C_VEL
LIN {X 0,Y 544.999,Z 352.247,A -85,B 0,C 180,E1 -3538.73,E2 -3538.73} C_VEL
LIN {X 0,Y 545.072,Z 346.331,A -85,B 0,C 180,E1 -3541.914,E2 -3541.914} C_VEL
LIN {X 0,Y 545.164,Z 341.518,A -85,B 0,C 180,E1 -3544.558,E2 -3544.558} C_VEL
LIN {X 0,Y 545.248,Z 336.607,A -85,B 0,C 180,E1 -3547.288,E2 -3547.288} C_VEL
LIN {X 0,Y 545.139,Z 333.211,A -85,B 0,C 180,E1 -3549.263,E2 -3549.263} C_VEL
LIN {X 0,Y 545.082,Z 333.212,A -85,B 0,C 180,E1 -3552.103,E2 -3552.103} C_VEL
LIN {X 0,Y 545.066,Z 333.214,A -85,B 0,C 180,E1 -3555.167,E2 -3555.167} C_VEL
LIN {X 0,Y 545.082,Z 333.213,A -85,B 0,C 180,E1 -3557.897,E2 -3557.897} C_VEL
LIN {X 0,Y 545.086,Z 333.209,A -85,B 0,C 180,E1 -3560.819,E2 -3560.819} C_VEL
LIN {X 0,Y 545.047,Z 333.216,A -85,B 0,C 180,E1 -3563.62,E2 -3563.62} C_VEL
LIN {X 0,Y 545.072,Z 333.215,A -85,B 0,C 180,E1 -3566.328,E2 -3566.328} C_VEL
LIN {X 0,Y 545.072,Z 333.211,A -85,B 0,C 180,E1 -3568.952,E2 -3568.952} C_VEL
LIN {X 0,Y 545.108,Z 333.213,A -85,B 0,C 180,E1 -3571.508,E2 -3571.508} C_VEL
LIN {X 0,Y 545.1,Z 333.208,A -85,B 0,C 180,E1 -3574.492,E2 -3574.492} C_VEL
LIN {X 0,Y 545.044,Z 333.215,A -85,B 0,C 180,E1 -3577.242,E2 -3577.242} C_VEL
LIN {X 0,Y 545.123,Z 333.207,A -85,B 0,C 180,E1 -3580.415,E2 -3580.415} C_VEL
LIN {X 0,Y 545.08,Z 333.214,A -85,B 0,C 180,E1 -3583.521,E2 -3583.521} C_VEL
LIN {X 0,Y 545.1,Z 333.207,A -85,B 0,C 180,E1 -3585.82,E2 -3585.82} C_VEL
LIN {X 0,Y 545.125,Z 333.206,A -85,B 0,C 180,E1 -3588.849,E2 -3588.849} C_VEL
LIN {X 0,Y 545.127,Z 333.21,A -85,B 0,C 180,E1 -3591.847,E2 -3591.847} C_VEL
LIN {X 0,Y 545.211,Z 333.196,A -85,B 0,C 180,E1 -3594.823,E2 -3594.823} C_VEL
LIN {X 0,Y 545.197,Z 333.195,A -85,B 0,C 180,E1 -3597.784,E2 -3597.784} C_VEL
LIN {X 0,Y 545.218,Z 333.193,A -85,B 0,C 180,E1 -3600.738,E2 -3600.738} C_VEL
LIN {X 0,Y 545.176,Z 333.199,A -85,B 0,C 180,E1 -3602.956,E2 -3602.956} C_VEL
LIN {X 0,Y 545.175,Z 333.198,A -85,B 0,C 180,E1 -3605.919,E2 -3605.919} C_VEL
LIN {X 0,Y 545.108,Z 333.21,A -85,B 0,C 180,E1 -3608.9,E2 -3608.9} C_VEL
LIN {X 0,Y 545.142,Z 333.209,A -85,B 0,C 180,E1 -3611.904,E2 -3611.904} C_VEL
LIN {X 0,Y 545.092,Z 333.212,A -85,B 0,C 180,E1 -3614.943,E2 -3614.943} C_VEL
LIN {X 0,Y 545.083,Z 333.211,A -85,B 0,C 180,E1 -3618.026,E2 -3618.026} C_VEL
LIN {X 0,Y 545.098,Z 333.215,A -85,B 0,C 180,E1 -3620.372,E2 -3620.372} C_VEL
LIN {X 0,Y 545.097,Z 333.213,A -85,B 0,C 180,E1 -3623.558,E2 -3623.558} C_VEL
LIN {X 0,Y 545.085,Z 333.21,A -85,B 0,C 180,E1 -3626,E2 -3626} C_VEL
LIN {X 0,Y 545.094,Z 333.215,A -85,B 0,C 180,E1 -3628.748,E2 -3628.748} C_VEL
LIN {X 0,Y 545.062,Z 333.215,A -85,B 0,C 180,E1 -3631.678,E2 -3631.678} C_VEL
LIN {X 0,Y 545.086,Z 333.21,A -85,B 0,C 180,E1 -3634.563,E2 -3634.563} C_VEL
LIN {X 0,Y 545.044,Z 333.22,A -85,B 0,C 180,E1 -3637.303,E2 -3637.303} C_VEL
LIN {X 0,Y 545.07,Z 333.214,A -85,B 0,C 180,E1 -3640.142,E2 -3640.142} C_VEL
LIN {X 0,Y 545.082,Z 333.212,A -85,B 0,C 180,E1 -3643.106,E2 -3643.106} C_VEL
LIN {X 0,Y 545.068,Z 333.214,A -85,B 0,C 180,E1 -3646.224,E2 -3646.224} C_VEL
LIN {X 0,Y 545.097,Z 333.215,A -85,B 0,C 180,E1 -3648.886,E2 -3648.886} C_VEL
LIN {X 0,Y 545.055,Z 333.219,A -85,B 0,C 180,E1 -3651.762,E2 -3651.762} C_VEL
LIN {X 0,Y 545.114,Z 333.43,A -85,B 0,C 180,E1 -3652.702,E2 -3652.702} C_VEL
LIN {X 0,Y 546.176,Z 339.189,A -85,B 0,C 180,E1 -3654.616,E2 -3654.616} C_VEL
LIN {X 0,Y 546.255,Z 345.064,A -85,B 0,C 180,E1 -3656.411,E2 -3656.411} C_VEL
LIN {X 0,Y 545.977,Z 355.221,A -85,B 0,C 180,E1 -3659.348,E2 -3659.348} C_VEL
LIN {X 0,Y 545.728,Z 366.084,A -85,B 0,C 180,E1 -3662.379,E2 -3662.379} C_VEL
LIN {X 0,Y 545.496,Z 376.681,A -85,B 0,C 180,E1 -3665.246,E2 -3665.246} C_VEL
LIN {X 0,Y 545.325,Z 387.601,A -85,B 0,C 180,E1 -3668.112,E2 -3668.112} C_VEL
LIN {X 0,Y 545.165,Z 397.951,A -85,B 0,C 180,E1 -3670.808,E2 -3670.808} C_VEL
LIN {X 0,Y 545.146,Z 400.444,A -85,B 0,C 180,E1 -3671.423,E2 -3671.423} C_VEL
LIN {X 0,Y 547.744,Z 411.935,A -85,B 0,C 180,E1 -3671.689,E2 -3671.689} C_VEL
LIN {X 0,Y 547.51,Z 427.694,A -85,B 0,C 180,E1 -3672.057,E2 -3672.057} C_VEL
LIN {X 0,Y 547.243,Z 442.665,A -85,B 0,C 180,E1 -3672.564,E2 -3672.564} C_VEL
LIN {X 0,Y 546.898,Z 456.773,A -85,B 0,C 180,E1 -3673.193,E2 -3673.193} C_VEL
LIN {X 0,Y 546.578,Z 470.247,A -85,B 0,C 180,E1 -3673.951,E2 -3673.951} C_VEL
LIN {X 0,Y 546.225,Z 482.553,A -85,B 0,C 180,E1 -3674.793,E2 -3674.793} C_VEL
LIN {X 0,Y 545.832,Z 495.29,A -85,B 0,C 180,E1 -3675.839,E2 -3675.839} C_VEL
LIN {X 0,Y 545.567,Z 506.748,A -85,B 0,C 180,E1 -3676.971,E2 -3676.971} C_VEL
LIN {X 0,Y 545.282,Z 516.388,A -85,B 0,C 180,E1 -3678.099,E2 -3678.099} C_VEL
LIN {X 0,Y 545.086,Z 525.854,A -85,B 0,C 180,E1 -3679.413,E2 -3679.413} C_VEL
LIN {X 0,Y 544.899,Z 533.734,A -85,B 0,C 180,E1 -3680.722,E2 -3680.722} C_VEL
LIN {X 0,Y 544.772,Z 541.089,A -85,B 0,C 180,E1 -3682.215,E2 -3682.215} C_VEL
LIN {X 0,Y 544.675,Z 546.916,A -85,B 0,C 180,E1 -3683.701,E2 -3683.701} C_VEL
LIN {X 0,Y 544.642,Z 550.386,A -85,B 0,C 180,E1 -3684.817,E2 -3684.817} C_VEL
LIN {X 0,Y 544.644,Z 553.888,A -85,B 0,C 180,E1 -3686.301,E2 -3686.301} C_VEL
LIN {X 0,Y 544.569,Z 556.191,A -85,B 0,C 180,E1 -3687.781,E2 -3687.781} C_VEL
LIN {X 0,Y 544.539,Z 557.348,A -85,B 0,C 180,E1 -3689.26,E2 -3689.26} C_VEL
LIN {X 0,Y 544.539,Z 557.348,A -85,B 0,C 180,E1 -3690.739,E2 -3690.739} C_VEL
LIN {X 0,Y 544.569,Z 556.188,A -85,B 0,C 180,E1 -3692.219,E2 -3692.219} C_VEL
LIN {X 0,Y 544.644,Z 553.885,A -85,B 0,C 180,E1 -3693.699,E2 -3693.699} C_VEL
LIN {X 0,Y 544.642,Z 550.387,A -85,B 0,C 180,E1 -3695.182,E2 -3695.182} C_VEL
LIN {X 0,Y 544.752,Z 545.609,A -85,B 0,C 180,E1 -3696.668,E2 -3696.668} C_VEL
LIN {X 0,Y 544.818,Z 539.421,A -85,B 0,C 180,E1 -3698.158,E2 -3698.158} C_VEL
LIN {X 0,Y 544.904,Z 531.645,A -85,B 0,C 180,E1 -3699.652,E2 -3699.652} C_VEL
LIN {X 0,Y 545.15,Z 523.367,A -85,B 0,C 180,E1 -3700.962,E2 -3700.962} C_VEL
LIN {X 0,Y 545.357,Z 513.391,A -85,B 0,C 180,E1 -3702.277,E2 -3702.277} C_VEL
LIN {X 0,Y 545.639,Z 503.186,A -85,B 0,C 180,E1 -3703.406,E2 -3703.406} C_VEL
LIN {X 0,Y 545.971,Z 491.018,A -85,B 0,C 180,E1 -3704.538,E2 -3704.538} C_VEL
LIN {X 0,Y 546.354,Z 478.644,A -85,B 0,C 180,E1 -3705.493,E2 -3705.493} C_VEL
LIN {X 0,Y 546.666,Z 465.507,A -85,B 0,C 180,E1 -3706.334,E2 -3706.334} C_VEL
LIN {X 0,Y 547.034,Z 450.823,A -85,B 0,C 180,E1 -3707.091,E2 -3707.091} C_VEL
LIN {X 0,Y 547.394,Z 435.844,A -85,B 0,C 180,E1 -3707.686,E2 -3707.686} C_VEL
LIN {X 0,Y 547.622,Z 420.72,A -85,B 0,C 180,E1 -3708.125,E2 -3708.125} C_VEL
LIN {X 0,Y 547.559,Z 410.77,A -85,B 0,C 180,E1 -3708.336,E2 -3708.336} C_VEL
LIN {X 0,Y 545.119,Z 400.288,A -85,B 0,C 180,E1 -3708.587,E2 -3708.587} C_VEL
LIN {X 0,Y 545.331,Z 389.003,A -85,B 0,C 180,E1 -3711.524,E2 -3711.524} C_VEL
LIN {X 0,Y 545.467,Z 378.196,A -85,B 0,C 180,E1 -3714.35,E2 -3714.35} C_VEL
LIN {X 0,Y 545.706,Z 367.262,A -85,B 0,C 180,E1 -3717.298,E2 -3717.298} C_VEL
LIN {X 0,Y 545.939,Z 356.116,A -85,B 0,C 180,E1 -3720.401,E2 -3720.401} C_VEL
LIN {X 0,Y 546.207,Z 346.254,A -85,B 0,C 180,E1 -3723.243,E2 -3723.243} C_VEL
LIN {X 0,Y 546.3,Z 340.597,A -85,B 0,C 180,E1 -3724.932,E2 -3724.932} C_VEL
LIN {X 0,Y 545.301,Z 334.429,A -85,B 0,C 180,E1 -3726.958,E2 -3726.958} C_VEL
LIN {X 0,Y 545.057,Z 333.22,A -85,B 0,C 180,E1 -3727.419,E2 -3727.419} C_VEL
LIN {X 0,Y 545.069,Z 333.215,A -85,B 0,C 180,E1 -3730.143,E2 -3730.143} C_VEL
LIN {X 0,Y 545.066,Z 333.218,A -85,B 0,C 180,E1 -3732.697,E2 -3732.697} C_VEL
LIN {X 0,Y 545.038,Z 333.217,A -85,B 0,C 180,E1 -3735.17,E2 -3735.17} C_VEL
LIN {X 0,Y 545.085,Z 333.214,A -85,B 0,C 180,E1 -3737.898,E2 -3737.898} C_VEL
LIN {X 0,Y 545.109,Z 333.208,A -85,B 0,C 180,E1 -3740.676,E2 -3740.676} C_VEL
LIN {X 0,Y 545.06,Z 333.214,A -85,B 0,C 180,E1 -3743.621,E2 -3743.621} C_VEL
LIN {X 0,Y 545.071,Z 333.218,A -85,B 0,C 180,E1 -3746.329,E2 -3746.329} C_VEL
LIN {X 0,Y 545.069,Z 333.213,A -85,B 0,C 180,E1 -3748.952,E2 -3748.952} C_VEL
LIN {X 0,Y 545.105,Z 333.211,A -85,B 0,C 180,E1 -3751.508,E2 -3751.508} C_VEL
LIN {X 0,Y 545.099,Z 333.212,A -85,B 0,C 180,E1 -3754.491,E2 -3754.491} C_VEL
LIN {X 0,Y 545.048,Z 333.214,A -85,B 0,C 180,E1 -3757.243,E2 -3757.243} C_VEL
LIN {X 0,Y 545.121,Z 333.205,A -85,B 0,C 180,E1 -3760.415,E2 -3760.415} C_VEL
LIN {X 0,Y 545.077,Z 333.211,A -85,B 0,C 180,E1 -3763.521,E2 -3763.521} C_VEL
LIN {X 0,Y 545.101,Z 333.208,A -85,B 0,C 180,E1 -3765.82,E2 -3765.82} C_VEL
LIN {X 0,Y 545.122,Z 333.205,A -85,B 0,C 180,E1 -3768.85,E2 -3768.85} C_VEL
LIN {X 0,Y 545.103,Z 333.21,A -85,B 0,C 180,E1 -3771.847,E2 -3771.847} C_VEL
LIN {X 0,Y 545.209,Z 333.2,A -85,B 0,C 180,E1 -3774.823,E2 -3774.823} C_VEL
LIN {X 0,Y 545.2,Z 333.195,A -85,B 0,C 180,E1 -3777.784,E2 -3777.784} C_VEL
LIN {X 0,Y 545.217,Z 333.191,A -85,B 0,C 180,E1 -3780.739,E2 -3780.739} C_VEL
LIN {X 0,Y 545.176,Z 333.201,A -85,B 0,C 180,E1 -3782.956,E2 -3782.956} C_VEL
LIN {X 0,Y 545.174,Z 333.198,A -85,B 0,C 180,E1 -3785.92,E2 -3785.92} C_VEL
LIN {X 0,Y 545.108,Z 333.207,A -85,B 0,C 180,E1 -3788.9,E2 -3788.9} C_VEL
LIN {X 0,Y 545.141,Z 333.206,A -85,B 0,C 180,E1 -3791.904,E2 -3791.904} C_VEL
LIN {X 0,Y 545.091,Z 333.214,A -85,B 0,C 180,E1 -3794.944,E2 -3794.944} C_VEL
LIN {X 0,Y 545.082,Z 333.211,A -85,B 0,C 180,E1 -3798.026,E2 -3798.026} C_VEL
LIN {X 0,Y 545.097,Z 333.21,A -85,B 0,C 180,E1 -3800.372,E2 -3800.372} C_VEL
LIN {X 0,Y 545.093,Z 333.212,A -85,B 0,C 180,E1 -3803.559,E2 -3803.559} C_VEL
LIN {X 0,Y 545.083,Z 333.21,A -85,B 0,C 180,E1 -3806.001,E2 -3806.001} C_VEL
LIN {X 0,Y 545.094,Z 333.211,A -85,B 0,C 180,E1 -3808.748,E2 -3808.748} C_VEL
LIN {X 0,Y 545.062,Z 333.217,A -85,B 0,C 180,E1 -3811.679,E2 -3811.679} C_VEL
LIN {X 0,Y 545.067,Z 333.212,A -85,B 0,C 180,E1 -3814.564,E2 -3814.564} C_VEL
LIN {X 0,Y 545.065,Z 333.217,A -85,B 0,C 180,E1 -3817.007,E2 -3817.007} C_VEL
LIN {X 0,Y 544.358,Z 333.302,A -85,B 0,C 180,E1 -3817.623,E2 -3817.623} C_VEL
LIN {X 0,Y 541.493,Z 333.663,A -85,B 0,C 180,E1 -3818.624,E2 -3818.624} C_VEL
LIN {X 0,Y 539.106,Z 333.957,A -85,B 0,C 180,E1 -3819.43,E2 -3819.43} C_VEL
LIN {X 0,Y 538.096,Z 334.085,A -85,B 0,C 180,E1 -3820.052,E2 -3820.052} C_VEL
LIN {X 0,Y 538.021,Z 334.089,A -85,B 0,C 180,E1 -3820.263,E2 -3820.263} C_VEL
LIN {X 0,Y 538.03,Z 334.089,A -85,B 0,C 180,E1 -3822.987,E2 -3822.987} C_VEL
LIN {X 0,Y 538.034,Z 334.09,A -85,B 0,C 180,E1 -3825.925,E2 -3825.925} C_VEL
LIN {X 0,Y 538.053,Z 334.089,A -85,B 0,C 180,E1 -3829.253,E2 -3829.253} C_VEL
LIN {X 0,Y 538.062,Z 334.137,A -85,B 0,C 180,E1 -3830.812,E2 -3830.812} C_VEL
LIN {X 0,Y 538.202,Z 338.118,A -85,B 0,C 180,E1 -3833.081,E2 -3833.081} C_VEL
LIN {X 0,Y 538.127,Z 343.015,A -85,B 0,C 180,E1 -3835.834,E2 -3835.834} C_VEL
LIN {X 0,Y 538.017,Z 347.839,A -85,B 0,C 180,E1 -3838.499,E2 -3838.499} C_VEL
LIN {X 0,Y 537.968,Z 352.613,A -85,B 0,C 180,E1 -3841.094,E2 -3841.094} C_VEL
LIN {X 0,Y 537.888,Z 357.379,A -85,B 0,C 180,E1 -3843.625,E2 -3843.625} C_VEL
LIN {X 0,Y 537.812,Z 362.246,A -85,B 0,C 180,E1 -3846.17,E2 -3846.17} C_VEL
LIN {X 0,Y 537.754,Z 366.854,A -85,B 0,C 180,E1 -3848.535,E2 -3848.535} C_VEL
LIN {X 0,Y 537.652,Z 373.122,A -85,B 0,C 180,E1 -3851.716,E2 -3851.716} C_VEL
LIN {X 0,Y 537.605,Z 377.523,A -85,B 0,C 180,E1 -3853.938,E2 -3853.938} C_VEL
LIN {X 0,Y 539.982,Z 388.842,A -85,B 0,C 180,E1 -3854.238,E2 -3854.238} C_VEL
LIN {X 0,Y 539.789,Z 402.129,A -85,B 0,C 180,E1 -3854.62,E2 -3854.62} C_VEL
LIN {X 0,Y 539.543,Z 416.218,A -85,B 0,C 180,E1 -3855.189,E2 -3855.189} C_VEL
LIN {X 0,Y 539.229,Z 428.892,A -85,B 0,C 180,E1 -3855.855,E2 -3855.855} C_VEL
LIN {X 0,Y 538.94,Z 440.532,A -85,B 0,C 180,E1 -3856.617,E2 -3856.617} C_VEL
LIN {X 0,Y 538.602,Z 452.381,A -85,B 0,C 180,E1 -3857.567,E2 -3857.567} C_VEL
LIN {X 0,Y 538.38,Z 462.596,A -85,B 0,C 180,E1 -3858.561,E2 -3858.561} C_VEL
LIN {X 0,Y 538.106,Z 471.986,A -85,B 0,C 180,E1 -3859.654,E2 -3859.654} C_VEL
LIN {X 0,Y 537.912,Z 480.111,A -85,B 0,C 180,E1 -3860.79,E2 -3860.79} C_VEL
LIN {X 0,Y 537.77,Z 487.891,A -85,B 0,C 180,E1 -3862.113,E2 -3862.113} C_VEL
LIN {X 0,Y 537.668,Z 494.101,A -85,B 0,C 180,E1 -3863.423,E2 -3863.423} C_VEL
LIN {X 0,Y 537.578,Z 499.053,A -85,B 0,C 180,E1 -3864.749,E2 -3864.749} C_VEL
LIN {X 0,Y 537.577,Z 503.211,A -85,B 0,C 180,E1 -3866.252,E2 -3866.252} C_VEL
LIN {X 0,Y 537.489,Z 505.937,A -85,B 0,C 180,E1 -3867.752,E2 -3867.752} C_VEL
LIN {X 0,Y 537.438,Z 507.307,A -85,B 0,C 180,E1 -3869.251,E2 -3869.251} C_VEL
LIN {X 0,Y 537.438,Z 507.354,A -85,B 0,C 180,E1 -3870.749,E2 -3870.749} C_VEL
LIN {X 0,Y 537.489,Z 506.072,A -85,B 0,C 180,E1 -3872.248,E2 -3872.248} C_VEL
LIN {X 0,Y 537.577,Z 503.426,A -85,B 0,C 180,E1 -3873.748,E2 -3873.748} C_VEL
LIN {X 0,Y 537.578,Z 499.347,A -85,B 0,C 180,E1 -3875.251,E2 -3875.251} C_VEL
LIN {X 0,Y 537.668,Z 493.719,A -85,B 0,C 180,E1 -3876.756,E2 -3876.756} C_VEL
LIN {X 0,Y 537.755,Z 487.367,A -85,B 0,C 180,E1 -3878.077,E2 -3878.077} C_VEL
LIN {X 0,Y 537.96,Z 479.464,A -85,B 0,C 180,E1 -3879.399,E2 -3879.399} C_VEL
LIN {X 0,Y 538.127,Z 471.202,A -85,B 0,C 180,E1 -3880.535,E2 -3880.535} C_VEL
LIN {X 0,Y 538.352,Z 462.093,A -85,B 0,C 180,E1 -3881.584,E2 -3881.584} C_VEL
LIN {X 0,Y 538.672,Z 451.241,A -85,B 0,C 180,E1 -3882.623,E2 -3882.623} C_VEL
LIN {X 0,Y 538.952,Z 439.151,A -85,B 0,C 180,E1 -3883.575,E2 -3883.575} C_VEL
LIN {X 0,Y 539.306,Z 427.201,A -85,B 0,C 180,E1 -3884.336,E2 -3884.336} C_VEL
LIN {X 0,Y 539.554,Z 414.005,A -85,B 0,C 180,E1 -3885.004,E2 -3885.004} C_VEL
LIN {X 0,Y 539.814,Z 400.4,A -85,B 0,C 180,E1 -3885.525,E2 -3885.525} C_VEL
LIN {X 0,Y 539.818,Z 388.022,A -85,B 0,C 180,E1 -3885.875,E2 -3885.875} C_VEL
LIN {X 0,Y 537.6,Z 377.522,A -85,B 0,C 180,E1 -3886.153,E2 -3886.153} C_VEL
LIN {X 0,Y 537.685,Z 371.742,A -85,B 0,C 180,E1 -3889.073,E2 -3889.073} C_VEL
LIN {X 0,Y 537.767,Z 365.458,A -85,B 0,C 180,E1 -3892.272,E2 -3892.272} C_VEL
LIN {X 0,Y 537.83,Z 360.726,A -85,B 0,C 180,E1 -3894.718,E2 -3894.718} C_VEL
LIN {X 0,Y 537.892,Z 355.764,A -85,B 0,C 180,E1 -3897.317,E2 -3897.317} C_VEL
LIN {X 0,Y 537.971,Z 351.18,A -85,B 0,C 180,E1 -3899.764,E2 -3899.764} C_VEL
LIN {X 0,Y 538.046,Z 346.403,A -85,B 0,C 180,E1 -3902.381,E2 -3902.381} C_VEL
LIN {X 0,Y 538.146,Z 341.566,A -85,B 0,C 180,E1 -3905.074,E2 -3905.074} C_VEL
LIN {X 0,Y 538.241,Z 336.621,A -85,B 0,C 180,E1 -3907.858,E2 -3907.858} C_VEL
LIN {X 0,Y 538.089,Z 334.089,A -85,B 0,C 180,E1 -3909.306,E2 -3909.306} C_VEL
LIN {X 0,Y 538.033,Z 334.092,A -85,B 0,C 180,E1 -3911.879,E2 -3911.879} C_VEL
LIN {X 0,Y 538.036,Z 334.093,A -85,B 0,C 180,E1 -3914.86,E2 -3914.86} C_VEL
LIN {X 0,Y 538.033,Z 334.093,A -85,B 0,C 180,E1 -3918.122,E2 -3918.122} C_VEL
LIN {X 0,Y 538.039,Z 334.087,A -85,B 0,C 180,E1 -3920.415,E2 -3920.415} C_VEL
LIN {X 0,Y 538.029,Z 334.093,A -85,B 0,C 180,E1 -3923.067,E2 -3923.067} C_VEL
LIN {X 0,Y 538.024,Z 334.089,A -85,B 0,C 180,E1 -3925.827,E2 -3925.827} C_VEL
LIN {X 0,Y 538.014,Z 334.094,A -85,B 0,C 180,E1 -3928.499,E2 -3928.499} C_VEL
LIN {X 0,Y 538.066,Z 334.085,A -85,B 0,C 180,E1 -3931.1,E2 -3931.1} C_VEL
LIN {X 0,Y 538.047,Z 334.088,A -85,B 0,C 180,E1 -3933.633,E2 -3933.633} C_VEL
LIN {X 0,Y 538.013,Z 334.091,A -85,B 0,C 180,E1 -3936.122,E2 -3936.122} C_VEL
LIN {X 0,Y 538.044,Z 334.086,A -85,B 0,C 180,E1 -3939.349,E2 -3939.349} C_VEL
LIN {X 0,Y 538.042,Z 334.086,A -85,B 0,C 180,E1 -3942.468,E2 -3942.468} C_VEL
LIN {X 0,Y 538.069,Z 334.084,A -85,B 0,C 180,E1 -3945.631,E2 -3945.631} C_VEL
LIN {X 0,Y 538.084,Z 334.084,A -85,B 0,C 180,E1 -3948.702,E2 -3948.702} C_VEL
LIN {X 0,Y 538.085,Z 334.086,A -85,B 0,C 180,E1 -3951.739,E2 -3951.739} C_VEL
LIN {X 0,Y 538.129,Z 334.076,A -85,B 0,C 180,E1 -3954.003,E2 -3954.003} C_VEL
LIN {X 0,Y 538.145,Z 334.077,A -85,B 0,C 180,E1 -3957.005,E2 -3957.005} C_VEL
LIN {X 0,Y 538.179,Z 334.074,A -85,B 0,C 180,E1 -3960,E2 -3960} C_VEL
LIN {X 0,Y 538.143,Z 334.075,A -85,B 0,C 180,E1 -3962.994,E2 -3962.994} C_VEL
LIN {X 0,Y 538.126,Z 334.076,A -85,B 0,C 180,E1 -3965.997,E2 -3965.997} C_VEL
LIN {X 0,Y 538.06,Z 334.086,A -85,B 0,C 180,E1 -3969.018,E2 -3969.018} C_VEL
LIN {X 0,Y 538.09,Z 334.087,A -85,B 0,C 180,E1 -3972.062,E2 -3972.062} C_VEL
LIN {X 0,Y 538.051,Z 334.091,A -85,B 0,C 180,E1 -3975.143,E2 -3975.143} C_VEL
LIN {X 0,Y 538.035,Z 334.091,A -85,B 0,C 180,E1 -3978.27,E2 -3978.27} C_VEL
LIN {X 0,Y 538.043,Z 334.091,A -85,B 0,C 180,E1 -3980.651,E2 -3980.651} C_VEL
LIN {X 0,Y 538.03,Z 334.093,A -85,B 0,C 180,E1 -3983.887,E2 -3983.887} C_VEL
LIN {X 0,Y 538.047,Z 334.087,A -85,B 0,C 180,E1 -3986.366,E2 -3986.366} C_VEL
LIN {X 0,Y 538.036,Z 334.091,A -85,B 0,C 180,E1 -3988.933,E2 -3988.933} C_VEL
LIN {X 0,Y 538.014,Z 334.096,A -85,B 0,C 180,E1 -3991.887,E2 -3991.887} C_VEL
LIN {X 0,Y 538.036,Z 334.089,A -85,B 0,C 180,E1 -3994.62,E2 -3994.62} C_VEL
LIN {X 0,Y 538.012,Z 334.097,A -85,B 0,C 180,E1 -3997.17,E2 -3997.17} C_VEL
LIN {X 0,Y 538.027,Z 334.089,A -85,B 0,C 180,E1 -3999.797,E2 -3999.797} C_VEL
LIN {X 0,Y 538.022,Z 334.092,A -85,B 0,C 180,E1 -4002.786,E2 -4002.786} C_VEL
LIN {X 0,Y 538.032,Z 334.092,A -85,B 0,C 180,E1 -4005.925,E2 -4005.925} C_VEL
LIN {X 0,Y 538.044,Z 334.089,A -85,B 0,C 180,E1 -4008.227,E2 -4008.227} C_VEL
LIN {X 0,Y 538.016,Z 334.095,A -85,B 0,C 180,E1 -4011.169,E2 -4011.169} C_VEL
LIN {X 0,Y 538.03,Z 334.18,A -85,B 0,C 180,E1 -4012.357,E2 -4012.357} C_VEL
LIN {X 0,Y 539.242,Z 340.64,A -85,B 0,C 180,E1 -4014.551,E2 -4014.551} C_VEL
LIN {X 0,Y 539.372,Z 345.035,A -85,B 0,C 180,E1 -4015.924,E2 -4015.924} C_VEL
LIN {X 0,Y 539.076,Z 355.487,A -85,B 0,C 180,E1 -4019.005,E2 -4019.005} C_VEL
LIN {X 0,Y 538.757,Z 366.008,A -85,B 0,C 180,E1 -4021.99,E2 -4021.99} C_VEL
LIN {X 0,Y 538.503,Z 376.561,A -85,B 0,C 180,E1 -4024.902,E2 -4024.902} C_VEL
LIN {X 0,Y 538.359,Z 385.694,A -85,B 0,C 180,E1 -4027.349,E2 -4027.349} C_VEL
LIN {X 0,Y 538.171,Z 397.939,A -85,B 0,C 180,E1 -4030.548,E2 -4030.548} C_VEL
LIN {X 0,Y 538.107,Z 400.45,A -85,B 0,C 180,E1 -4031.171,E2 -4031.171} C_VEL
LIN {X 0,Y 540.952,Z 412.554,A -85,B 0,C 180,E1 -4031.463,E2 -4031.463} C_VEL
LIN {X 0,Y 540.746,Z 428.28,A -85,B 0,C 180,E1 -4031.843,E2 -4031.843} C_VEL
LIN {X 0,Y 540.461,Z 442.95,A -85,B 0,C 180,E1 -4032.35,E2 -4032.35} C_VEL
LIN {X 0,Y 540.071,Z 456.775,A -85,B 0,C 180,E1 -4032.974,E2 -4032.974} C_VEL
LIN {X 0,Y 539.723,Z 470.249,A -85,B 0,C 180,E1 -4033.742,E2 -4033.742} C_VEL
LIN {X 0,Y 539.315,Z 483.278,A -85,B 0,C 180,E1 -4034.648,E2 -4034.648} C_VEL
LIN {X 0,Y 538.902,Z 495.288,A -85,B 0,C 180,E1 -4035.653,E2 -4035.653} C_VEL
LIN {X 0,Y 538.593,Z 506.747,A -85,B 0,C 180,E1 -4036.8,E2 -4036.8} C_VEL
LIN {X 0,Y 538.283,Z 516.387,A -85,B 0,C 180,E1 -4037.942,E2 -4037.942} C_VEL
LIN {X 0,Y 538.068,Z 525.853,A -85,B 0,C 180,E1 -4039.273,E2 -4039.273} C_VEL
LIN {X 0,Y 537.824,Z 533.734,A -85,B 0,C 180,E1 -4040.599,E2 -4040.599} C_VEL
LIN {X 0,Y 537.699,Z 541.089,A -85,B 0,C 180,E1 -4042.112,E2 -4042.112} C_VEL
LIN {X 0,Y 537.627,Z 546.39,A -85,B 0,C 180,E1 -4043.459,E2 -4043.459} C_VEL
LIN {X 0,Y 537.574,Z 550.386,A -85,B 0,C 180,E1 -4044.749,E2 -4044.749} C_VEL
LIN {X 0,Y 537.561,Z 553.888,A -85,B 0,C 180,E1 -4046.252,E2 -4046.252} C_VEL
LIN {X 0,Y 537.488,Z 556.19,A -85,B 0,C 180,E1 -4047.752,E2 -4047.752} C_VEL
LIN {X 0,Y 537.44,Z 557.348,A -85,B 0,C 180,E1 -4049.251,E2 -4049.251} C_VEL
LIN {X 0,Y 537.44,Z 557.347,A -85,B 0,C 180,E1 -4050.749,E2 -4050.749} C_VEL
LIN {X 0,Y 537.488,Z 556.187,A -85,B 0,C 180,E1 -4052.248,E2 -4052.248} C_VEL
LIN {X 0,Y 537.561,Z 553.884,A -85,B 0,C 180,E1 -4053.748,E2 -4053.748} C_VEL
LIN {X 0,Y 537.574,Z 550.387,A -85,B 0,C 180,E1 -4055.251,E2 -4055.251} C_VEL
LIN {X 0,Y 537.664,Z 545.609,A -85,B 0,C 180,E1 -4056.756,E2 -4056.756} C_VEL
LIN {X 0,Y 537.734,Z 539.421,A -85,B 0,C 180,E1 -4058.266,E2 -4058.266} C_VEL
LIN {X 0,Y 537.859,Z 531.644,A -85,B 0,C 180,E1 -4059.78,E2 -4059.78} C_VEL
LIN {X 0,Y 538.102,Z 523.367,A -85,B 0,C 180,E1 -4061.107,E2 -4061.107} C_VEL
LIN {X 0,Y 538.358,Z 513.391,A -85,B 0,C 180,E1 -4062.439,E2 -4062.439} C_VEL
LIN {X 0,Y 538.662,Z 503.185,A -85,B 0,C 180,E1 -4063.583,E2 -4063.583} C_VEL
LIN {X 0,Y 539.022,Z 491.018,A -85,B 0,C 180,E1 -4064.729,E2 -4064.729} C_VEL
LIN {X 0,Y 539.473,Z 478.826,A -85,B 0,C 180,E1 -4065.682,E2 -4065.682} C_VEL
LIN {X 0,Y 539.81,Z 465.504,A -85,B 0,C 180,E1 -4066.547,E2 -4066.547} C_VEL
LIN {X 0,Y 540.234,Z 450.821,A -85,B 0,C 180,E1 -4067.313,E2 -4067.313} C_VEL
LIN {X 0,Y 540.612,Z 436.427,A -85,B 0,C 180,E1 -4067.893,E2 -4067.893} C_VEL
LIN {X 0,Y 540.851,Z 421.989,A -85,B 0,C 180,E1 -4068.326,E2 -4068.326} C_VEL
LIN {X 0,Y 540.917,Z 412.33,A -85,B 0,C 180,E1 -4068.543,E2 -4068.543} C_VEL
LIN {X 0,Y 538.096,Z 400.261,A -85,B 0,C 180,E1 -4068.846,E2 -4068.846} C_VEL
LIN {X 0,Y 538.3,Z 389.146,A -85,B 0,C 180,E1 -4071.739,E2 -4071.739} C_VEL
LIN {X 0,Y 538.443,Z 379.536,A -85,B 0,C 180,E1 -4074.292,E2 -4074.292} C_VEL
LIN {X 0,Y 538.734,Z 367.86,A -85,B 0,C 180,E1 -4077.491,E2 -4077.491} C_VEL
LIN {X 0,Y 538.993,Z 356.797,A -85,B 0,C 180,E1 -4080.618,E2 -4080.618} C_VEL
LIN {X 0,Y 539.29,Z 347.018,A -85,B 0,C 180,E1 -4083.484,E2 -4083.484} C_VEL
LIN {X 0,Y 539.372,Z 342.088,A -85,B 0,C 180,E1 -4084.982,E2 -4084.982} C_VEL
LIN {X 0,Y 538.293,Z 335.412,A -85,B 0,C 180,E1 -4087.21,E2 -4087.21} C_VEL
LIN {X 0,Y 538.019,Z 334.097,A -85,B 0,C 180,E1 -4087.69,E2 -4087.69} C_VEL
LIN {X 0,Y 538.052,Z 334.091,A -85,B 0,C 180,E1 -4090.776,E2 -4090.776} C_VEL
LIN {X 0,Y 538.032,Z 334.088,A -85,B 0,C 180,E1 -4094.075,E2 -4094.075} C_VEL
LIN {X 0,Y 538.021,Z 334.091,A -85,B 0,C 180,E1 -4097.214,E2 -4097.214} C_VEL
LIN {X 0,Y 538.057,Z 334.086,A -85,B 0,C 180,E1 -4100.206,E2 -4100.206} C_VEL
LIN {X 0,Y 538.033,Z 334.094,A -85,B 0,C 180,E1 -4103.068,E2 -4103.068} C_VEL
LIN {X 0,Y 538.03,Z 334.092,A -85,B 0,C 180,E1 -4105.828,E2 -4105.828} C_VEL
LIN {X 0,Y 538.012,Z 334.093,A -85,B 0,C 180,E1 -4108.499,E2 -4108.499} C_VEL
LIN {X 0,Y 538.064,Z 334.089,A -85,B 0,C 180,E1 -4111.1,E2 -4111.1} C_VEL
LIN {X 0,Y 538.046,Z 334.087,A -85,B 0,C 180,E1 -4113.634,E2 -4113.634} C_VEL
LIN {X 0,Y 538.027,Z 334.093,A -85,B 0,C 180,E1 -4116.118,E2 -4116.118} C_VEL
LIN {X 0,Y 538.042,Z 334.088,A -85,B 0,C 180,E1 -4119.349,E2 -4119.349} C_VEL
LIN {X 0,Y 538.059,Z 334.085,A -85,B 0,C 180,E1 -4122.517,E2 -4122.517} C_VEL
LIN {X 0,Y 538.069,Z 334.083,A -85,B 0,C 180,E1 -4125.631,E2 -4125.631} C_VEL
LIN {X 0,Y 538.082,Z 334.083,A -85,B 0,C 180,E1 -4128.702,E2 -4128.702} C_VEL
LIN {X 0,Y 538.067,Z 334.087,A -85,B 0,C 180,E1 -4131.739,E2 -4131.739} C_VEL
LIN {X 0,Y 538.128,Z 334.075,A -85,B 0,C 180,E1 -4134.003,E2 -4134.003} C_VEL
LIN {X 0,Y 538.142,Z 334.074,A -85,B 0,C 180,E1 -4137.006,E2 -4137.006} C_VEL
LIN {X 0,Y 538.179,Z 334.073,A -85,B 0,C 180,E1 -4140,E2 -4140} C_VEL
LIN {X 0,Y 538.143,Z 334.078,A -85,B 0,C 180,E1 -4142.995,E2 -4142.995} C_VEL
LIN {X 0,Y 538.128,Z 334.077,A -85,B 0,C 180,E1 -4145.997,E2 -4145.997} C_VEL
LIN {X 0,Y 538.061,Z 334.084,A -85,B 0,C 180,E1 -4149.018,E2 -4149.018} C_VEL
LIN {X 0,Y 538.089,Z 334.083,A -85,B 0,C 180,E1 -4152.063,E2 -4152.063} C_VEL
LIN {X 0,Y 538.051,Z 334.091,A -85,B 0,C 180,E1 -4155.144,E2 -4155.144} C_VEL
LIN {X 0,Y 538.034,Z 334.092,A -85,B 0,C 180,E1 -4158.27,E2 -4158.27} C_VEL
LIN {X 0,Y 538.042,Z 334.086,A -85,B 0,C 180,E1 -4160.651,E2 -4160.651} C_VEL
LIN {X 0,Y 538.03,Z 334.088,A -85,B 0,C 180,E1 -4163.887,E2 -4163.887} C_VEL
LIN {X 0,Y 538.046,Z 334.088,A -85,B 0,C 180,E1 -4166.367,E2 -4166.367} C_VEL
LIN {X 0,Y 538.036,Z 334.088,A -85,B 0,C 180,E1 -4168.933,E2 -4168.933} C_VEL
LIN {X 0,Y 538.015,Z 334.096,A -85,B 0,C 180,E1 -4171.887,E2 -4171.887} C_VEL
LIN {X 0,Y 538.017,Z 334.091,A -85,B 0,C 180,E1 -4174.618,E2 -4174.618} C_VEL
LIN {X 0,Y 538.008,Z 334.094,A -85,B 0,C 180,E1 -4177.17,E2 -4177.17} C_VEL
LIN {X 0,Y 538.021,Z 334.089,A -85,B 0,C 180,E1 -4180.263,E2 -4180.263} C_VEL
LIN {X 0,Y 537.371,Z 334.173,A -85,B 0,C 180,E1 -4180.888,E2 -4180.888} C_VEL
LIN {X 0,Y 534.52,Z 334.533,A -85,B 0,C 180,E1 -4181.903,E2 -4181.903} C_VEL
LIN {X 0,Y 532.095,Z 334.837,A -85,B 0,C 180,E1 -4182.72,E2 -4182.72} C_VEL
LIN {X 0,Y 531.048,Z 334.965,A -85,B 0,C 180,E1 -4183.351,E2 -4183.351} C_VEL
LIN {X 0,Y 530.961,Z 334.973,A -85,B 0,C 180,E1 -4183.565,E2 -4183.565} C_VEL
LIN {X 0,Y 530.969,Z 334.971,A -85,B 0,C 180,E1 -4186.505,E2 -4186.505} C_VEL
LIN {X 0,Y 530.985,Z 334.969,A -85,B 0,C 180,E1 -4189.567,E2 -4189.567} C_VEL
LIN {X 0,Y 531.05,Z 335.138,A -85,B 0,C 180,E1 -4190.767,E2 -4190.767} C_VEL
LIN {X 0,Y 531.18,Z 338.206,A -85,B 0,C 180,E1 -4192.548,E2 -4192.548} C_VEL
LIN {X 0,Y 531.1,Z 343.062,A -85,B 0,C 180,E1 -4195.318,E2 -4195.318} C_VEL
LIN {X 0,Y 531.007,Z 347.915,A -85,B 0,C 180,E1 -4198.034,E2 -4198.034} C_VEL
LIN {X 0,Y 530.909,Z 353.101,A -85,B 0,C 180,E1 -4200.89,E2 -4200.89} C_VEL
LIN {X 0,Y 530.84,Z 357.474,A -85,B 0,C 180,E1 -4203.247,E2 -4203.247} C_VEL
LIN {X 0,Y 530.75,Z 362.718,A -85,B 0,C 180,E1 -4206.018,E2 -4206.018} C_VEL
LIN {X 0,Y 530.671,Z 368.559,A -85,B 0,C 180,E1 -4209.048,E2 -4209.048} C_VEL
LIN {X 0,Y 530.605,Z 374.851,A -85,B 0,C 180,E1 -4212.263,E2 -4212.263} C_VEL
LIN {X 0,Y 530.561,Z 377.631,A -85,B 0,C 180,E1 -4213.676,E2 -4213.676} C_VEL
LIN {X 0,Y 533.204,Z 390.233,A -85,B 0,C 180,E1 -4214.042,E2 -4214.042} C_VEL
LIN {X 0,Y 532.992,Z 403.139,A -85,B 0,C 180,E1 -4214.428,E2 -4214.428} C_VEL
LIN {X 0,Y 532.728,Z 416.749,A -85,B 0,C 180,E1 -4214.995,E2 -4214.995} C_VEL
LIN {X 0,Y 532.375,Z 429.254,A -85,B 0,C 180,E1 -4215.669,E2 -4215.669} C_VEL
LIN {X 0,Y 532.025,Z 440.744,A -85,B 0,C 180,E1 -4216.439,E2 -4216.439} C_VEL
LIN {X 0,Y 531.644,Z 452.444,A -85,B 0,C 180,E1 -4217.401,E2 -4217.401} C_VEL
LIN {X 0,Y 531.325,Z 463.976,A -85,B 0,C 180,E1 -4218.556,E2 -4218.556} C_VEL
LIN {X 0,Y 531.028,Z 473.475,A -85,B 0,C 180,E1 -4219.708,E2 -4219.708} C_VEL
LIN {X 0,Y 530.811,Z 482.537,A -85,B 0,C 180,E1 -4221.05,E2 -4221.05} C_VEL
LIN {X 0,Y 530.643,Z 489.838,A -85,B 0,C 180,E1 -4222.389,E2 -4222.389} C_VEL
LIN {X 0,Y 530.559,Z 496.4,A -85,B 0,C 180,E1 -4223.917,E2 -4223.917} C_VEL
LIN {X 0,Y 530.449,Z 501.319,A -85,B 0,C 180,E1 -4225.441,E2 -4225.441} C_VEL
LIN {X 0,Y 530.453,Z 504.748,A -85,B 0,C 180,E1 -4226.962,E2 -4226.962} C_VEL
LIN {X 0,Y 530.36,Z 506.789,A -85,B 0,C 180,E1 -4228.481,E2 -4228.481} C_VEL
LIN {X 0,Y 530.342,Z 507.497,A -85,B 0,C 180,E1 -4230,E2 -4230} C_VEL
LIN {X 0,Y 530.358,Z 506.88,A -85,B 0,C 180,E1 -4231.519,E2 -4231.519} C_VEL
LIN {X 0,Y 530.452,Z 504.923,A -85,B 0,C 180,E1 -4233.038,E2 -4233.038} C_VEL
LIN {X 0,Y 530.449,Z 501.57,A -85,B 0,C 180,E1 -4234.56,E2 -4234.56} C_VEL
LIN {X 0,Y 530.537,Z 496.733,A -85,B 0,C 180,E1 -4236.084,E2 -4236.084} C_VEL
LIN {X 0,Y 530.587,Z 492.075,A -85,B 0,C 180,E1 -4237.229,E2 -4237.229} C_VEL
LIN {X 0,Y 530.774,Z 485.296,A -85,B 0,C 180,E1 -4238.567,E2 -4238.567} C_VEL
LIN {X 0,Y 530.915,Z 476.87,A -85,B 0,C 180,E1 -4239.909,E2 -4239.909} C_VEL
LIN {X 0,Y 531.222,Z 468.084,A -85,B 0,C 180,E1 -4241.06,E2 -4241.06} C_VEL
LIN {X 0,Y 531.473,Z 457.432,A -85,B 0,C 180,E1 -4242.215,E2 -4242.215} C_VEL
LIN {X 0,Y 531.809,Z 446.798,A -85,B 0,C 180,E1 -4243.177,E2 -4243.177} C_VEL
LIN {X 0,Y 532.177,Z 435.182,A -85,B 0,C 180,E1 -4244.044,E2 -4244.044} C_VEL
LIN {X 0,Y 532.556,Z 422.365,A -85,B 0,C 180,E1 -4244.814,E2 -4244.814} C_VEL
LIN {X 0,Y 532.873,Z 410.893,A -85,B 0,C 180,E1 -4245.358,E2 -4245.358} C_VEL
LIN {X 0,Y 533.069,Z 397.008,A -85,B 0,C 180,E1 -4245.863,E2 -4245.863} C_VEL
LIN {X 0,Y 533.115,Z 389.464,A -85,B 0,C 180,E1 -4246.072,E2 -4246.072} C_VEL
LIN {X 0,Y 530.556,Z 377.648,A -85,B 0,C 180,E1 -4246.399,E2 -4246.399} C_VEL
LIN {X 0,Y 530.614,Z 371.905,A -85,B 0,C 180,E1 -4249.337,E2 -4249.337} C_VEL
LIN {X 0,Y 530.693,Z 366.654,A -85,B 0,C 180,E1 -4252.025,E2 -4252.025} C_VEL
LIN {X 0,Y 530.767,Z 360.823,A -85,B 0,C 180,E1 -4255.07,E2 -4255.07} C_VEL
LIN {X 0,Y 530.852,Z 356.044,A -85,B 0,C 180,E1 -4257.605,E2 -4257.605} C_VEL
LIN {X 0,Y 530.953,Z 350.464,A -85,B 0,C 180,E1 -4260.641,E2 -4260.641} C_VEL
LIN {X 0,Y 531.072,Z 344.865,A -85,B 0,C 180,E1 -4263.767,E2 -4263.767} C_VEL
LIN {X 0,Y 531.179,Z 339.97,A -85,B 0,C 180,E1 -4266.541,E2 -4266.541} C_VEL
LIN {X 0,Y 531.11,Z 335.297,A -85,B 0,C 180,E1 -4269.228,E2 -4269.228} C_VEL
LIN {X 0,Y 531.043,Z 334.968,A -85,B 0,C 180,E1 -4269.439,E2 -4269.439} C_VEL
LIN {X 0,Y 530.982,Z 334.969,A -85,B 0,C 180,E1 -4272.457,E2 -4272.457} C_VEL
LIN {X 0,Y 530.99,Z 334.966,A -85,B 0,C 180,E1 -4275.453,E2 -4275.453} C_VEL
LIN {X 0,Y 530.998,Z 334.965,A -85,B 0,C 180,E1 -4278.565,E2 -4278.565} C_VEL
LIN {X 0,Y 530.963,Z 334.974,A -85,B 0,C 180,E1 -4281.53,E2 -4281.53} C_VEL
LIN {X 0,Y 530.96,Z 334.97,A -85,B 0,C 180,E1 -4284.38,E2 -4284.38} C_VEL
LIN {X 0,Y 530.972,Z 334.968,A -85,B 0,C 180,E1 -4287.134,E2 -4287.134} C_VEL
LIN {X 0,Y 530.976,Z 334.972,A -85,B 0,C 180,E1 -4289.803,E2 -4289.803} C_VEL
LIN {X 0,Y 531.019,Z 334.962,A -85,B 0,C 180,E1 -4292.468,E2 -4292.468} C_VEL
LIN {X 0,Y 531.011,Z 334.969,A -85,B 0,C 180,E1 -4294.943,E2 -4294.943} C_VEL
LIN {X 0,Y 530.978,Z 334.973,A -85,B 0,C 180,E1 -4298.247,E2 -4298.247} C_VEL
LIN {X 0,Y 530.998,Z 334.965,A -85,B 0,C 180,E1 -4300.677,E2 -4300.677} C_VEL
LIN {X 0,Y 530.982,Z 334.969,A -85,B 0,C 180,E1 -4303.071,E2 -4303.071} C_VEL
LIN {X 0,Y 531.025,Z 334.962,A -85,B 0,C 180,E1 -4305.436,E2 -4305.436} C_VEL
LIN {X 0,Y 531.044,Z 334.963,A -85,B 0,C 180,E1 -4308.55,E2 -4308.55} C_VEL
LIN {X 0,Y 531.055,Z 334.961,A -85,B 0,C 180,E1 -4311.629,E2 -4311.629} C_VEL
LIN {X 0,Y 531.127,Z 334.949,A -85,B 0,C 180,E1 -4314.685,E2 -4314.685} C_VEL
LIN {X 0,Y 531.142,Z 334.946,A -85,B 0,C 180,E1 -4317.725,E2 -4317.725} C_VEL
LIN {X 0,Y 531.159,Z 334.944,A -85,B 0,C 180,E1 -4320.758,E2 -4320.758} C_VEL
LIN {X 0,Y 531.109,Z 334.952,A -85,B 0,C 180,E1 -4323.034,E2 -4323.034} C_VEL
LIN {X 0,Y 531.082,Z 334.954,A -85,B 0,C 180,E1 -4326.077,E2 -4326.077} C_VEL
LIN {X 0,Y 531.022,Z 334.963,A -85,B 0,C 180,E1 -4329.138,E2 -4329.138} C_VEL
LIN {X 0,Y 531.047,Z 334.962,A -85,B 0,C 180,E1 -4332.225,E2 -4332.225} C_VEL
LIN {X 0,Y 531.001,Z 334.971,A -85,B 0,C 180,E1 -4335.349,E2 -4335.349} C_VEL
LIN {X 0,Y 530.994,Z 334.971,A -85,B 0,C 180,E1 -4338.521,E2 -4338.521} C_VEL
LIN {X 0,Y 531.004,Z 334.965,A -85,B 0,C 180,E1 -4340.938,E2 -4340.938} C_VEL
LIN {X 0,Y 530.986,Z 334.967,A -85,B 0,C 180,E1 -4344.224,E2 -4344.224} C_VEL
LIN {X 0,Y 531.007,Z 334.967,A -85,B 0,C 180,E1 -4346.743,E2 -4346.743} C_VEL
LIN {X 0,Y 530.986,Z 334.966,A -85,B 0,C 180,E1 -4349.322,E2 -4349.322} C_VEL
LIN {X 0,Y 530.97,Z 334.974,A -85,B 0,C 180,E1 -4352.1,E2 -4352.1} C_VEL
LIN {X 0,Y 530.993,Z 334.967,A -85,B 0,C 180,E1 -4354.854,E2 -4354.854} C_VEL
LIN {X 0,Y 530.971,Z 334.971,A -85,B 0,C 180,E1 -4357.507,E2 -4357.507} C_VEL
LIN {X 0,Y 530.985,Z 334.972,A -85,B 0,C 180,E1 -4360.432,E2 -4360.432} C_VEL
LIN {X 0,Y 530.964,Z 334.972,A -85,B 0,C 180,E1 -4363.281,E2 -4363.281} C_VEL
LIN {X 0,Y 530.985,Z 334.973,A -85,B 0,C 180,E1 -4365.621,E2 -4365.621} C_VEL
LIN {X 0,Y 531.003,Z 334.969,A -85,B 0,C 180,E1 -4368.565,E2 -4368.565} C_VEL
LIN {X 0,Y 530.96,Z 334.974,A -85,B 0,C 180,E1 -4371.529,E2 -4371.529} C_VEL
LIN {X 0,Y 530.997,Z 335.126,A -85,B 0,C 180,E1 -4372.075,E2 -4372.075} C_VEL
LIN {X 0,Y 532.135,Z 340.934,A -85,B 0,C 180,E1 -4374.095,E2 -4374.095} C_VEL
LIN {X 0,Y 532.486,Z 345.021,A -85,B 0,C 180,E1 -4375.421,E2 -4375.421} C_VEL
LIN {X 0,Y 532.161,Z 355.431,A -85,B 0,C 180,E1 -4378.556,E2 -4378.556} C_VEL
LIN {X 0,Y 531.786,Z 365.936,A -85,B 0,C 180,E1 -4381.59,E2 -4381.59} C_VEL
LIN {X 0,Y 531.535,Z 376.46,A -85,B 0,C 180,E1 -4384.55,E2 -4384.55} C_VEL
LIN {X 0,Y 531.312,Z 387.072,A -85,B 0,C 180,E1 -4387.443,E2 -4387.443} C_VEL
LIN {X 0,Y 531.135,Z 397.89,A -85,B 0,C 180,E1 -4390.319,E2 -4390.319} C_VEL
LIN {X 0,Y 531.062,Z 400.215,A -85,B 0,C 180,E1 -4390.924,E2 -4390.924} C_VEL
LIN {X 0,Y 534.222,Z 414.199,A -85,B 0,C 180,E1 -4391.264,E2 -4391.264} C_VEL
LIN {X 0,Y 533.967,Z 429.601,A -85,B 0,C 180,E1 -4391.651,E2 -4391.651} C_VEL
LIN {X 0,Y 533.689,Z 443.173,A -85,B 0,C 180,E1 -4392.128,E2 -4392.128} C_VEL
LIN {X 0,Y 533.262,Z 456.778,A -85,B 0,C 180,E1 -4392.75,E2 -4392.75} C_VEL
LIN {X 0,Y 532.86,Z 470.249,A -85,B 0,C 180,E1 -4393.526,E2 -4393.526} C_VEL
LIN {X 0,Y 532.447,Z 482.98,A -85,B 0,C 180,E1 -4394.423,E2 -4394.423} C_VEL
LIN {X 0,Y 531.975,Z 495.286,A -85,B 0,C 180,E1 -4395.462,E2 -4395.462} C_VEL
LIN {X 0,Y 531.608,Z 506.746,A -85,B 0,C 180,E1 -4396.623,E2 -4396.623} C_VEL
LIN {X 0,Y 531.286,Z 516.387,A -85,B 0,C 180,E1 -4397.781,E2 -4397.781} C_VEL
LIN {X 0,Y 531.052,Z 525.852,A -85,B 0,C 180,E1 -4399.13,E2 -4399.13} C_VEL
LIN {X 0,Y 530.764,Z 533.734,A -85,B 0,C 180,E1 -4400.473,E2 -4400.473} C_VEL
LIN {X 0,Y 530.64,Z 541.089,A -85,B 0,C 180,E1 -4402.006,E2 -4402.006} C_VEL
LIN {X 0,Y 530.545,Z 546.698,A -85,B 0,C 180,E1 -4403.466,E2 -4403.466} C_VEL
LIN {X 0,Y 530.509,Z 550.386,A -85,B 0,C 180,E1 -4404.679,E2 -4404.679} C_VEL
LIN {X 0,Y 530.48,Z 553.887,A -85,B 0,C 180,E1 -4406.202,E2 -4406.202} C_VEL
LIN {X 0,Y 530.409,Z 556.19,A -85,B 0,C 180,E1 -4407.722,E2 -4407.722} C_VEL
LIN {X 0,Y 530.342,Z 557.348,A -85,B 0,C 180,E1 -4409.241,E2 -4409.241} C_VEL
LIN {X 0,Y 530.342,Z 557.347,A -85,B 0,C 180,E1 -4410.759,E2 -4410.759} C_VEL
LIN {X 0,Y 530.409,Z 556.187,A -85,B 0,C 180,E1 -4412.278,E2 -4412.278} C_VEL
LIN {X 0,Y 530.48,Z 553.884,A -85,B 0,C 180,E1 -4413.798,E2 -4413.798} C_VEL
LIN {X 0,Y 530.509,Z 550.387,A -85,B 0,C 180,E1 -4415.321,E2 -4415.321} C_VEL
LIN {X 0,Y 530.569,Z 545.609,A -85,B 0,C 180,E1 -4416.847,E2 -4416.847} C_VEL
LIN {X 0,Y 530.665,Z 539.42,A -85,B 0,C 180,E1 -4418.377,E2 -4418.377} C_VEL
LIN {X 0,Y 530.809,Z 531.643,A -85,B 0,C 180,E1 -4419.911,E2 -4419.911} C_VEL
LIN {X 0,Y 531.057,Z 523.366,A -85,B 0,C 180,E1 -4421.256,E2 -4421.256} C_VEL
LIN {X 0,Y 531.383,Z 513.391,A -85,B 0,C 180,E1 -4422.605,E2 -4422.605} C_VEL
LIN {X 0,Y 531.707,Z 503.184,A -85,B 0,C 180,E1 -4423.764,E2 -4423.764} C_VEL
LIN {X 0,Y 532.121,Z 491.017,A -85,B 0,C 180,E1 -4424.925,E2 -4424.925} C_VEL
LIN {X 0,Y 532.61,Z 477.59,A -85,B 0,C 180,E1 -4425.981,E2 -4425.981} C_VEL
LIN {X 0,Y 533.083,Z 463.879,A -85,B 0,C 180,E1 -4426.86,E2 -4426.86} C_VEL
LIN {X 0,Y 533.471,Z 449.799,A -85,B 0,C 180,E1 -4427.589,E2 -4427.589} C_VEL
LIN {X 0,Y 533.879,Z 434.578,A -85,B 0,C 180,E1 -4428.192,E2 -4428.192} C_VEL
LIN {X 0,Y 534.151,Z 419.149,A -85,B 0,C 180,E1 -4428.632,E2 -4428.632} C_VEL
LIN {X 0,Y 534.142,Z 413.36,A -85,B 0,C 180,E1 -4428.757,E2 -4428.757} C_VEL
LIN {X 0,Y 531.05,Z 400.145,A -85,B 0,C 180,E1 -4429.096,E2 -4429.096} C_VEL
LIN {X 0,Y 531.278,Z 390.104,A -85,B 0,C 180,E1 -4431.74,E2 -4431.74} C_VEL
LIN {X 0,Y 531.439,Z 379.469,A -85,B 0,C 180,E1 -4434.618,E2 -4434.618} C_VEL
LIN {X 0,Y 531.76,Z 368.48,A -85,B 0,C 180,E1 -4437.687,E2 -4437.687} C_VEL
LIN {X 0,Y 532.114,Z 356.92,A -85,B 0,C 180,E1 -4441.004,E2 -4441.004} C_VEL
LIN {X 0,Y 532.452,Z 346.499,A -85,B 0,C 180,E1 -4444.123,E2 -4444.123} C_VEL
LIN {X 0,Y 532.293,Z 342.089,A -85,B 0,C 180,E1 -4445.517,E2 -4445.517} C_VEL
LIN {X 0,Y 530.967,Z 334.976,A -85,B 0,C 180,E1 -4447.987,E2 -4447.987} C_VEL
LIN {X 0,Y 530.99,Z 334.97,A -85,B 0,C 180,E1 -4451.024,E2 -4451.024} C_VEL
LIN {X 0,Y 530.967,Z 334.966,A -85,B 0,C 180,E1 -4453.495,E2 -4453.495} C_VEL
LIN {X 0,Y 530.957,Z 334.974,A -85,B 0,C 180,E1 -4456.505,E2 -4456.505} C_VEL
LIN {X 0,Y 531.029,Z 334.964,A -85,B 0,C 180,E1 -4459.572,E2 -4459.572} C_VEL
LIN {X 0,Y 530.972,Z 334.971,A -85,B 0,C 180,E1 -4462.577,E2 -4462.577} C_VEL
LIN {X 0,Y 531.005,Z 334.966,A -85,B 0,C 180,E1 -4465.311,E2 -4465.311} C_VEL
LIN {X 0,Y 530.97,Z 334.974,A -85,B 0,C 180,E1 -4468.032,E2 -4468.032} C_VEL
LIN {X 0,Y 530.992,Z 334.967,A -85,B 0,C 180,E1 -4470.874,E2 -4470.874} C_VEL
LIN {X 0,Y 531.006,Z 334.967,A -85,B 0,C 180,E1 -4473.257,E2 -4473.257} C_VEL
LIN {X 0,Y 531.002,Z 334.966,A -85,B 0,C 180,E1 -4475.958,E2 -4475.958} C_VEL
LIN {X 0,Y 531.003,Z 334.963,A -85,B 0,C 180,E1 -4479.062,E2 -4479.062} C_VEL
LIN {X 0,Y 530.993,Z 334.97,A -85,B 0,C 180,E1 -4481.479,E2 -4481.479} C_VEL
LIN {X 0,Y 531,Z 334.967,A -85,B 0,C 180,E1 -4484.651,E2 -4484.651} C_VEL
LIN {X 0,Y 531.046,Z 334.959,A -85,B 0,C 180,E1 -4487.775,E2 -4487.775} C_VEL
LIN {X 0,Y 531.021,Z 334.961,A -85,B 0,C 180,E1 -4490.862,E2 -4490.862} C_VEL
LIN {X 0,Y 531.088,Z 334.952,A -85,B 0,C 180,E1 -4493.923,E2 -4493.923} C_VEL
LIN {X 0,Y 531.109,Z 334.951,A -85,B 0,C 180,E1 -4496.966,E2 -4496.966} C_VEL
LIN {X 0,Y 531.15,Z 334.949,A -85,B 0,C 180,E1 -4500,E2 -4500} C_VEL
LIN {X 0,Y 531.109,Z 334.954,A -85,B 0,C 180,E1 -4503.034,E2 -4503.034} C_VEL
LIN {X 0,Y 531.088,Z 334.954,A -85,B 0,C 180,E1 -4506.077,E2 -4506.077} C_VEL
LIN {X 0,Y 531.054,Z 334.962,A -85,B 0,C 180,E1 -4508.371,E2 -4508.371} C_VEL
LIN {X 0,Y 531.072,Z 334.959,A -85,B 0,C 180,E1 -4511.68,E2 -4511.68} C_VEL
LIN {X 0,Y 531.036,Z 334.964,A -85,B 0,C 180,E1 -4514.956,E2 -4514.956} C_VEL
LIN {X 0,Y 531.022,Z 334.961,A -85,B 0,C 180,E1 -4517.722,E2 -4517.722} C_VEL
LIN {X 0,Y 531.03,Z 334.966,A -85,B 0,C 180,E1 -4520.127,E2 -4520.127} C_VEL
LIN {X 0,Y 530.969,Z 334.974,A -85,B 0,C 180,E1 -4523.396,E2 -4523.396} C_VEL
LIN {X 0,Y 531.018,Z 334.962,A -85,B 0,C 180,E1 -4525.897,E2 -4525.897} C_VEL
LIN {X 0,Y 531.001,Z 334.97,A -85,B 0,C 180,E1 -4528.455,E2 -4528.455} C_VEL
LIN {X 0,Y 530.962,Z 334.969,A -85,B 0,C 180,E1 -4531.079,E2 -4531.079} C_VEL
LIN {X 0,Y 530.991,Z 334.969,A -85,B 0,C 180,E1 -4533.773,E2 -4533.773} C_VEL
LIN {X 0,Y 530.959,Z 334.972,A -85,B 0,C 180,E1 -4536.558,E2 -4536.558} C_VEL
LIN {X 0,Y 530.99,Z 334.966,A -85,B 0,C 180,E1 -4539.443,E2 -4539.443} C_VEL
LIN {X 0,Y 530.982,Z 334.968,A -85,B 0,C 180,E1 -4542.457,E2 -4542.457} C_VEL
LIN {X 0,Y 530.961,Z 334.973,A -85,B 0,C 180,E1 -4543.565,E2 -4543.565} C_VEL
LIN {X 0,Y 530.29,Z 335.055,A -85,B 0,C 180,E1 -4544.198,E2 -4544.198} C_VEL
LIN {X 0,Y 527.445,Z 335.413,A -85,B 0,C 180,E1 -4545.227,E2 -4545.227} C_VEL
LIN {X 0,Y 525.042,Z 335.716,A -85,B 0,C 180,E1 -4546.056,E2 -4546.056} C_VEL
LIN {X 0,Y 524.009,Z 335.843,A -85,B 0,C 180,E1 -4546.695,E2 -4546.695} C_VEL
LIN {X 0,Y 523.924,Z 335.851,A -85,B 0,C 180,E1 -4546.912,E2 -4546.912} C_VEL
LIN {X 0,Y 523.952,Z 335.847,A -85,B 0,C 180,E1 -4549.921,E2 -4549.921} C_VEL
LIN {X 0,Y 524.015,Z 336.064,A -85,B 0,C 180,E1 -4550.675,E2 -4550.675} C_VEL
LIN {X 0,Y 524.153,Z 339.824,A -85,B 0,C 180,E1 -4552.888,E2 -4552.888} C_VEL
LIN {X 0,Y 524.049,Z 344.751,A -85,B 0,C 180,E1 -4555.718,E2 -4555.718} C_VEL
LIN {X 0,Y 523.939,Z 349.6,A -85,B 0,C 180,E1 -4558.457,E2 -4558.457} C_VEL
LIN {X 0,Y 523.853,Z 354.385,A -85,B 0,C 180,E1 -4561.12,E2 -4561.12} C_VEL
LIN {X 0,Y 523.759,Z 359.739,A -85,B 0,C 180,E1 -4564.031,E2 -4564.031} C_VEL
LIN {X 0,Y 523.668,Z 365.509,A -85,B 0,C 180,E1 -4567.095,E2 -4567.095} C_VEL
LIN {X 0,Y 523.554,Z 371.091,A -85,B 0,C 180,E1 -4569.994,E2 -4569.994} C_VEL
LIN {X 0,Y 523.539,Z 376.638,A -85,B 0,C 180,E1 -4572.823,E2 -4572.823} C_VEL
LIN {X 0,Y 523.512,Z 378.022,A -85,B 0,C 180,E1 -4573.45,E2 -4573.45} C_VEL
LIN {X 0,Y 526.411,Z 390.624,A -85,B 0,C 180,E1 -4573.812,E2 -4573.812} C_VEL
LIN {X 0,Y 526.2,Z 404.33,A -85,B 0,C 180,E1 -4574.235,E2 -4574.235} C_VEL
LIN {X 0,Y 525.923,Z 417.509,A -85,B 0,C 180,E1 -4574.796,E2 -4574.796} C_VEL
LIN {X 0,Y 525.557,Z 429.939,A -85,B 0,C 180,E1 -4575.479,E2 -4575.479} C_VEL
LIN {X 0,Y 525.149,Z 441.376,A -85,B 0,C 180,E1 -4576.258,E2 -4576.258} C_VEL
LIN {X 0,Y 524.733,Z 453.03,A -85,B 0,C 180,E1 -4577.233,E2 -4577.233} C_VEL
LIN {X 0,Y 524.38,Z 463.031,A -85,B 0,C 180,E1 -4578.246,E2 -4578.246} C_VEL
LIN {X 0,Y 524.096,Z 472.312,A -85,B 0,C 180,E1 -4579.375,E2 -4579.375} C_VEL
LIN {X 0,Y 523.862,Z 480.305,A -85,B 0,C 180,E1 -4580.541,E2 -4580.541} C_VEL
LIN {X 0,Y 523.654,Z 487.966,A -85,B 0,C 180,E1 -4581.899,E2 -4581.899} C_VEL
LIN {X 0,Y 523.488,Z 494.972,A -85,B 0,C 180,E1 -4583.452,E2 -4583.452} C_VEL
LIN {X 0,Y 523.451,Z 499.057,A -85,B 0,C 180,E1 -4584.607,E2 -4584.607} C_VEL
LIN {X 0,Y 523.419,Z 503.213,A -85,B 0,C 180,E1 -4586.151,E2 -4586.151} C_VEL
LIN {X 0,Y 523.334,Z 505.938,A -85,B 0,C 180,E1 -4587.691,E2 -4587.691} C_VEL
LIN {X 0,Y 523.246,Z 507.309,A -85,B 0,C 180,E1 -4589.23,E2 -4589.23} C_VEL
LIN {X 0,Y 523.247,Z 507.354,A -85,B 0,C 180,E1 -4590.77,E2 -4590.77} C_VEL
LIN {X 0,Y 523.333,Z 506.071,A -85,B 0,C 180,E1 -4592.309,E2 -4592.309} C_VEL
LIN {X 0,Y 523.419,Z 503.424,A -85,B 0,C 180,E1 -4593.85,E2 -4593.85} C_VEL
LIN {X 0,Y 523.448,Z 499.342,A -85,B 0,C 180,E1 -4595.393,E2 -4595.393} C_VEL
LIN {X 0,Y 523.496,Z 493.713,A -85,B 0,C 180,E1 -4596.94,E2 -4596.94} C_VEL
LIN {X 0,Y 523.684,Z 486.444,A -85,B 0,C 180,E1 -4598.489,E2 -4598.489} C_VEL
LIN {X 0,Y 523.87,Z 478.434,A -85,B 0,C 180,E1 -4599.849,E2 -4599.849} C_VEL
LIN {X 0,Y 524.198,Z 470.049,A -85,B 0,C 180,E1 -4601.014,E2 -4601.014} C_VEL
LIN {X 0,Y 524.527,Z 459.82,A -85,B 0,C 180,E1 -4602.191,E2 -4602.191} C_VEL
LIN {X 0,Y 524.897,Z 448.551,A -85,B 0,C 180,E1 -4603.256,E2 -4603.256} C_VEL
LIN {X 0,Y 525.319,Z 435.827,A -85,B 0,C 180,E1 -4604.231,E2 -4604.231} C_VEL
LIN {X 0,Y 525.749,Z 423.066,A -85,B 0,C 180,E1 -4605.011,E2 -4605.011} C_VEL
LIN {X 0,Y 526.076,Z 411.847,A -85,B 0,C 180,E1 -4605.554,E2 -4605.554} C_VEL
LIN {X 0,Y 526.313,Z 397.489,A -85,B 0,C 180,E1 -4606.086,E2 -4606.086} C_VEL
LIN {X 0,Y 526.273,Z 390.093,A -85,B 0,C 180,E1 -4606.298,E2 -4606.298} C_VEL
LIN {X 0,Y 523.491,Z 377.758,A -85,B 0,C 180,E1 -4606.652,E2 -4606.652} C_VEL
LIN {X 0,Y 523.575,Z 372.068,A -85,B 0,C 180,E1 -4609.608,E2 -4609.608} C_VEL
LIN {X 0,Y 523.669,Z 365.688,A -85,B 0,C 180,E1 -4612.905,E2 -4612.905} C_VEL
LIN {X 0,Y 523.756,Z 359.91,A -85,B 0,C 180,E1 -4615.968,E2 -4615.968} C_VEL
LIN {X 0,Y 523.842,Z 354.544,A -85,B 0,C 180,E1 -4618.881,E2 -4618.881} C_VEL
LIN {X 0,Y 523.937,Z 349.755,A -85,B 0,C 180,E1 -4621.543,E2 -4621.543} C_VEL
LIN {X 0,Y 524.048,Z 344.913,A -85,B 0,C 180,E1 -4624.282,E2 -4624.282} C_VEL
LIN {X 0,Y 524.173,Z 340.004,A -85,B 0,C 180,E1 -4627.111,E2 -4627.111} C_VEL
LIN {X 0,Y 523.998,Z 335.846,A -85,B 0,C 180,E1 -4629.575,E2 -4629.575} C_VEL
LIN {X 0,Y 523.939,Z 335.846,A -85,B 0,C 180,E1 -4632.459,E2 -4632.459} C_VEL
LIN {X 0,Y 523.958,Z 335.842,A -85,B 0,C 180,E1 -4635.309,E2 -4635.309} C_VEL
LIN {X 0,Y 523.96,Z 335.841,A -85,B 0,C 180,E1 -4638.69,E2 -4638.69} C_VEL
LIN {X 0,Y 523.923,Z 335.846,A -85,B 0,C 180,E1 -4641.081,E2 -4641.081} C_VEL
LIN {X 0,Y 523.905,Z 335.848,A -85,B 0,C 180,E1 -4643.825,E2 -4643.825} C_VEL
LIN {X 0,Y 523.947,Z 335.848,A -85,B 0,C 180,E1 -4646.636,E2 -4646.636} C_VEL
LIN {X 0,Y 523.961,Z 335.842,A -85,B 0,C 180,E1 -4649.356,E2 -4649.356} C_VEL
LIN {X 0,Y 523.983,Z 335.839,A -85,B 0,C 180,E1 -4652.282,E2 -4652.282} C_VEL
LIN {X 0,Y 523.958,Z 335.842,A -85,B 0,C 180,E1 -4654.581,E2 -4654.581} C_VEL
LIN {X 0,Y 523.918,Z 335.848,A -85,B 0,C 180,E1 -4657.107,E2 -4657.107} C_VEL
LIN {X 0,Y 523.985,Z 335.841,A -85,B 0,C 180,E1 -4659.866,E2 -4659.866} C_VEL
LIN {X 0,Y 523.964,Z 335.841,A -85,B 0,C 180,E1 -4662.837,E2 -4662.837} C_VEL
LIN {X 0,Y 523.983,Z 335.842,A -85,B 0,C 180,E1 -4665.236,E2 -4665.236} C_VEL
LIN {X 0,Y 524.019,Z 335.838,A -85,B 0,C 180,E1 -4668.394,E2 -4668.394} C_VEL
LIN {X 0,Y 524.003,Z 335.838,A -85,B 0,C 180,E1 -4671.516,E2 -4671.516} C_VEL
LIN {X 0,Y 524.088,Z 335.825,A -85,B 0,C 180,E1 -4674.614,E2 -4674.614} C_VEL
LIN {X 0,Y 524.115,Z 335.821,A -85,B 0,C 180,E1 -4677.694,E2 -4677.694} C_VEL
LIN {X 0,Y 524.129,Z 335.82,A -85,B 0,C 180,E1 -4680.768,E2 -4680.768} C_VEL
LIN {X 0,Y 524.076,Z 335.828,A -85,B 0,C 180,E1 -4683.075,E2 -4683.075} C_VEL
LIN {X 0,Y 524.044,Z 335.831,A -85,B 0,C 180,E1 -4686.159,E2 -4686.159} C_VEL
LIN {X 0,Y 523.992,Z 335.838,A -85,B 0,C 180,E1 -4689.262,E2 -4689.262} C_VEL
LIN {X 0,Y 524.032,Z 335.836,A -85,B 0,C 180,E1 -4691.751,E2 -4691.751} C_VEL
LIN {X 0,Y 523.999,Z 335.84,A -85,B 0,C 180,E1 -4695.052,E2 -4695.052} C_VEL
LIN {X 0,Y 523.969,Z 335.841,A -85,B 0,C 180,E1 -4697.969,E2 -4697.969} C_VEL
LIN {X 0,Y 523.977,Z 335.846,A -85,B 0,C 180,E1 -4700.41,E2 -4700.41} C_VEL
LIN {X 0,Y 523.923,Z 335.846,A -85,B 0,C 180,E1 -4702.893,E2 -4702.893} C_VEL
LIN {X 0,Y 523.959,Z 335.847,A -85,B 0,C 180,E1 -4705.418,E2 -4705.418} C_VEL
LIN {X 0,Y 523.973,Z 335.84,A -85,B 0,C 180,E1 -4707.999,E2 -4707.999} C_VEL
LIN {X 0,Y 523.949,Z 335.845,A -85,B 0,C 180,E1 -4710.854,E2 -4710.854} C_VEL
LIN {X 0,Y 523.966,Z 335.847,A -85,B 0,C 180,E1 -4713.734,E2 -4713.734} C_VEL
LIN {X 0,Y 523.927,Z 335.847,A -85,B 0,C 180,E1 -4716.404,E2 -4716.404} C_VEL
LIN {X 0,Y 523.924,Z 335.848,A -85,B 0,C 180,E1 -4719.084,E2 -4719.084} C_VEL
LIN {X 0,Y 523.957,Z 335.849,A -85,B 0,C 180,E1 -4722.118,E2 -4722.118} C_VEL
LIN {X 0,Y 523.949,Z 335.845,A -85,B 0,C 180,E1 -4725.309,E2 -4725.309} C_VEL
LIN {X 0,Y 523.964,Z 335.846,A -85,B 0,C 180,E1 -4728.689,E2 -4728.689} C_VEL
LIN {X 0,Y 523.948,Z 336.039,A -85,B 0,C 180,E1 -4731.778,E2 -4731.778} C_VEL
LIN {X 0,Y 525.147,Z 342.097,A -85,B 0,C 180,E1 -4733.924,E2 -4733.924} C_VEL
LIN {X 0,Y 525.562,Z 346.484,A -85,B 0,C 180,E1 -4735.366,E2 -4735.366} C_VEL
LIN {X 0,Y 525.195,Z 356.87,A -85,B 0,C 180,E1 -4738.541,E2 -4738.541} C_VEL
LIN {X 0,Y 524.801,Z 367.364,A -85,B 0,C 180,E1 -4741.614,E2 -4741.614} C_VEL
LIN {X 0,Y 524.526,Z 377.886,A -85,B 0,C 180,E1 -4744.611,E2 -4744.611} C_VEL
LIN {X 0,Y 524.273,Z 388.857,A -85,B 0,C 180,E1 -4747.662,E2 -4747.662} C_VEL
LIN {X 0,Y 524.037,Z 400.126,A -85,B 0,C 180,E1 -4750.687,E2 -4750.687} C_VEL
LIN {X 0,Y 527.418,Z 415.181,A -85,B 0,C 180,E1 -4751.062,E2 -4751.062} C_VEL
LIN {X 0,Y 527.1,Z 430.986,A -85,B 0,C 180,E1 -4751.48,E2 -4751.48} C_VEL
LIN {X 0,Y 526.719,Z 446.168,A -85,B 0,C 180,E1 -4752.05,E2 -4752.05} C_VEL
LIN {X 0,Y 526.295,Z 459.842,A -85,B 0,C 180,E1 -4752.715,E2 -4752.715} C_VEL
LIN {X 0,Y 525.832,Z 474.324,A -85,B 0,C 180,E1 -4753.6,E2 -4753.6} C_VEL
LIN {X 0,Y 525.362,Z 487.421,A -85,B 0,C 180,E1 -4754.581,E2 -4754.581} C_VEL
LIN {X 0,Y 524.888,Z 499.322,A -85,B 0,C 180,E1 -4755.658,E2 -4755.658} C_VEL
LIN {X 0,Y 524.511,Z 510.136,A -85,B 0,C 180,E1 -4756.833,E2 -4756.833} C_VEL
LIN {X 0,Y 524.14,Z 519.309,A -85,B 0,C 180,E1 -4758.005,E2 -4758.005} C_VEL
LIN {X 0,Y 523.943,Z 528.295,A -85,B 0,C 180,E1 -4759.371,E2 -4759.371} C_VEL
LIN {X 0,Y 523.699,Z 535.748,A -85,B 0,C 180,E1 -4760.733,E2 -4760.733} C_VEL
LIN {X 0,Y 523.535,Z 542.699,A -85,B 0,C 180,E1 -4762.285,E2 -4762.285} C_VEL
LIN {X 0,Y 523.441,Z 548.162,A -85,B 0,C 180,E1 -4763.834,E2 -4763.834} C_VEL
LIN {X 0,Y 523.322,Z 552.29,A -85,B 0,C 180,E1 -4765.378,E2 -4765.378} C_VEL
LIN {X 0,Y 523.358,Z 555.184,A -85,B 0,C 180,E1 -4766.921,E2 -4766.921} C_VEL
LIN {X 0,Y 523.272,Z 556.909,A -85,B 0,C 180,E1 -4768.461,E2 -4768.461} C_VEL
LIN {X 0,Y 523.243,Z 557.5,A -85,B 0,C 180,E1 -4770,E2 -4770} C_VEL
LIN {X 0,Y 523.272,Z 556.907,A -85,B 0,C 180,E1 -4771.539,E2 -4771.539} C_VEL
LIN {X 0,Y 523.358,Z 555.18,A -85,B 0,C 180,E1 -4773.079,E2 -4773.079} C_VEL
LIN {X 0,Y 523.322,Z 552.288,A -85,B 0,C 180,E1 -4774.622,E2 -4774.622} C_VEL
LIN {X 0,Y 523.451,Z 548.165,A -85,B 0,C 180,E1 -4776.166,E2 -4776.166} C_VEL
LIN {X 0,Y 523.535,Z 542.701,A -85,B 0,C 180,E1 -4777.715,E2 -4777.715} C_VEL
LIN {X 0,Y 523.699,Z 535.743,A -85,B 0,C 180,E1 -4779.267,E2 -4779.267} C_VEL
LIN {X 0,Y 523.987,Z 527.08,A -85,B 0,C 180,E1 -4780.823,E2 -4780.823} C_VEL
LIN {X 0,Y 524.232,Z 517.846,A -85,B 0,C 180,E1 -4782.193,E2 -4782.193} C_VEL
LIN {X 0,Y 524.598,Z 508.507,A -85,B 0,C 180,E1 -4783.362,E2 -4783.362} C_VEL
LIN {X 0,Y 525.011,Z 496.359,A -85,B 0,C 180,E1 -4784.635,E2 -4784.635} C_VEL
LIN {X 0,Y 525.456,Z 484.823,A -85,B 0,C 180,E1 -4785.634,E2 -4785.634} C_VEL
LIN {X 0,Y 525.924,Z 471.436,A -85,B 0,C 180,E1 -4786.597,E2 -4786.597} C_VEL
LIN {X 0,Y 526.35,Z 458.047,A -85,B 0,C 180,E1 -4787.383,E2 -4787.383} C_VEL
LIN {X 0,Y 526.804,Z 444.386,A -85,B 0,C 180,E1 -4788.026,E2 -4788.026} C_VEL
LIN {X 0,Y 527.137,Z 429.433,A -85,B 0,C 180,E1 -4788.569,E2 -4788.569} C_VEL
LIN {X 0,Y 527.376,Z 414.617,A -85,B 0,C 180,E1 -4788.951,E2 -4788.951} C_VEL
LIN {X 0,Y 524.047,Z 400.075,A -85,B 0,C 180,E1 -4789.327,E2 -4789.327} C_VEL
LIN {X 0,Y 524.273,Z 388.862,A -85,B 0,C 180,E1 -4792.338,E2 -4792.338} C_VEL
LIN {X 0,Y 524.53,Z 377.881,A -85,B 0,C 180,E1 -4795.389,E2 -4795.389} C_VEL
LIN {X 0,Y 524.809,Z 367.353,A -85,B 0,C 180,E1 -4798.386,E2 -4798.386} C_VEL
LIN {X 0,Y 525.201,Z 356.855,A -85,B 0,C 180,E1 -4801.459,E2 -4801.459} C_VEL
LIN {X 0,Y 525.602,Z 346.482,A -85,B 0,C 180,E1 -4804.631,E2 -4804.631} C_VEL
LIN {X 0,Y 524.883,Z 340.726,A -85,B 0,C 180,E1 -4806.546,E2 -4806.546} C_VEL
LIN {X 0,Y 523.924,Z 335.853,A -85,B 0,C 180,E1 -4808.346,E2 -4808.346} C_VEL
LIN {X 0,Y 523.963,Z 335.843,A -85,B 0,C 180,E1 -4811.311,E2 -4811.311} C_VEL
LIN {X 0,Y 523.948,Z 335.849,A -85,B 0,C 180,E1 -4814.69,E2 -4814.69} C_VEL
LIN {X 0,Y 523.959,Z 335.845,A -85,B 0,C 180,E1 -4817.882,E2 -4817.882} C_VEL
LIN {X 0,Y 523.963,Z 335.845,A -85,B 0,C 180,E1 -4820.919,E2 -4820.919} C_VEL
LIN {X 0,Y 523.932,Z 335.846,A -85,B 0,C 180,E1 -4823.828,E2 -4823.828} C_VEL
LIN {X 0,Y 523.945,Z 335.847,A -85,B 0,C 180,E1 -4826.636,E2 -4826.636} C_VEL
LIN {X 0,Y 523.959,Z 335.846,A -85,B 0,C 180,E1 -4829.356,E2 -4829.356} C_VEL
LIN {X 0,Y 523.98,Z 335.839,A -85,B 0,C 180,E1 -4832.282,E2 -4832.282} C_VEL
LIN {X 0,Y 523.958,Z 335.846,A -85,B 0,C 180,E1 -4834.582,E2 -4834.582} C_VEL
LIN {X 0,Y 523.921,Z 335.846,A -85,B 0,C 180,E1 -4837.107,E2 -4837.107} C_VEL
LIN {X 0,Y 523.983,Z 335.843,A -85,B 0,C 180,E1 -4839.866,E2 -4839.866} C_VEL
LIN {X 0,Y 523.971,Z 335.843,A -85,B 0,C 180,E1 -4842.838,E2 -4842.838} C_VEL
LIN {X 0,Y 523.982,Z 335.839,A -85,B 0,C 180,E1 -4845.236,E2 -4845.236} C_VEL
LIN {X 0,Y 524.02,Z 335.837,A -85,B 0,C 180,E1 -4848.394,E2 -4848.394} C_VEL
LIN {X 0,Y 523.993,Z 335.843,A -85,B 0,C 180,E1 -4851.516,E2 -4851.516} C_VEL
LIN {X 0,Y 524.05,Z 335.829,A -85,B 0,C 180,E1 -4853.841,E2 -4853.841} C_VEL
LIN {X 0,Y 524.075,Z 335.827,A -85,B 0,C 180,E1 -4856.925,E2 -4856.925} C_VEL
LIN {X 0,Y 524.12,Z 335.824,A -85,B 0,C 180,E1 -4860,E2 -4860} C_VEL
LIN {X 0,Y 524.076,Z 335.831,A -85,B 0,C 180,E1 -4863.075,E2 -4863.075} C_VEL
LIN {X 0,Y 524.051,Z 335.831,A -85,B 0,C 180,E1 -4866.159,E2 -4866.159} C_VEL
LIN {X 0,Y 524.002,Z 335.84,A -85,B 0,C 180,E1 -4868.484,E2 -4868.484} C_VEL
LIN {X 0,Y 524.031,Z 335.837,A -85,B 0,C 180,E1 -4871.751,E2 -4871.751} C_VEL
LIN {X 0,Y 523.999,Z 335.84,A -85,B 0,C 180,E1 -4875.052,E2 -4875.052} C_VEL
LIN {X 0,Y 523.969,Z 335.841,A -85,B 0,C 180,E1 -4877.969,E2 -4877.969} C_VEL
LIN {X 0,Y 523.977,Z 335.84,A -85,B 0,C 180,E1 -4880.41,E2 -4880.41} C_VEL
LIN {X 0,Y 523.92,Z 335.847,A -85,B 0,C 180,E1 -4882.893,E2 -4882.893} C_VEL
LIN {X 0,Y 523.958,Z 335.844,A -85,B 0,C 180,E1 -4885.419,E2 -4885.419} C_VEL
LIN {X 0,Y 523.973,Z 335.84,A -85,B 0,C 180,E1 -4887.999,E2 -4887.999} C_VEL
LIN {X 0,Y 523.949,Z 335.843,A -85,B 0,C 180,E1 -4890.855,E2 -4890.855} C_VEL
LIN {X 0,Y 523.963,Z 335.845,A -85,B 0,C 180,E1 -4893.734,E2 -4893.734} C_VEL
LIN {X 0,Y 523.907,Z 335.849,A -85,B 0,C 180,E1 -4896.401,E2 -4896.401} C_VEL
LIN {X 0,Y 523.924,Z 335.847,A -85,B 0,C 180,E1 -4899.085,E2 -4899.085} C_VEL
LIN {X 0,Y 523.955,Z 335.846,A -85,B 0,C 180,E1 -4902.119,E2 -4902.119} C_VEL
LIN {X 0,Y 523.96,Z 335.848,A -85,B 0,C 180,E1 -4905.309,E2 -4905.309} C_VEL
LIN {X 0,Y 523.924,Z 335.851,A -85,B 0,C 180,E1 -4906.912,E2 -4906.912} C_VEL
LIN {X 0,Y 523.261,Z 335.932,A -85,B 0,C 180,E1 -4907.553,E2 -4907.553} C_VEL
LIN {X 0,Y 520.437,Z 336.286,A -85,B 0,C 180,E1 -4908.595,E2 -4908.595} C_VEL
LIN {X 0,Y 518.046,Z 336.584,A -85,B 0,C 180,E1 -4909.434,E2 -4909.434} C_VEL
LIN {X 0,Y 517.015,Z 336.712,A -85,B 0,C 180,E1 -4910.082,E2 -4910.082} C_VEL
LIN {X 0,Y 516.928,Z 336.723,A -85,B 0,C 180,E1 -4910.301,E2 -4910.301} C_VEL
LIN {X 0,Y 517.13,Z 339.851,A -85,B 0,C 180,E1 -4912.297,E2 -4912.297} C_VEL
LIN {X 0,Y 517.04,Z 344.8,A -85,B 0,C 180,E1 -4915.187,E2 -4915.187} C_VEL
LIN {X 0,Y 516.924,Z 349.681,A -85,B 0,C 180,E1 -4917.978,E2 -4917.978} C_VEL
LIN {X 0,Y 516.816,Z 354.481,A -85,B 0,C 180,E1 -4920.689,E2 -4920.689} C_VEL
LIN {X 0,Y 516.703,Z 359.255,A -85,B 0,C 180,E1 -4923.33,E2 -4923.33} C_VEL
LIN {X 0,Y 516.662,Z 364.023,A -85,B 0,C 180,E1 -4925.916,E2 -4925.916} C_VEL
LIN {X 0,Y 516.533,Z 368.821,A -85,B 0,C 180,E1 -4928.447,E2 -4928.447} C_VEL
LIN {X 0,Y 516.465,Z 373.616,A -85,B 0,C 180,E1 -4930.938,E2 -4930.938} C_VEL
LIN {X 0,Y 516.447,Z 378.112,A -85,B 0,C 180,E1 -4933.191,E2 -4933.191} C_VEL
LIN {X 0,Y 519.63,Z 391.679,A -85,B 0,C 180,E1 -4933.594,E2 -4933.594} C_VEL
LIN {X 0,Y 519.436,Z 405.194,A -85,B 0,C 180,E1 -4934.024,E2 -4934.024} C_VEL
LIN {X 0,Y 519.129,Z 418.27,A -85,B 0,C 180,E1 -4934.592,E2 -4934.592} C_VEL
LIN {X 0,Y 518.719,Z 430.627,A -85,B 0,C 180,E1 -4935.283,E2 -4935.283} C_VEL
LIN {X 0,Y 518.291,Z 442.007,A -85,B 0,C 180,E1 -4936.073,E2 -4936.073} C_VEL
LIN {X 0,Y 517.853,Z 453.614,A -85,B 0,C 180,E1 -4937.06,E2 -4937.06} C_VEL
LIN {X 0,Y 517.44,Z 463.874,A -85,B 0,C 180,E1 -4938.12,E2 -4938.12} C_VEL
